// TIA Portal project "Assembler" (V17)

(* hardware
DEVICE "S7-1500/ET200MP station_1"  S7-1500 station
   slot 0: "Rail_0"  Rack  6ES7 590-1***0-0AA0
   slot 1: "PLC_1"  CPU 1511-1 PN  6ES7 511-1AK02-0AB0  V2.9
      slot 3: "CPU display_1"  6ES7591-1AA00-0AA0
      slot 32768: "PROFINET interface_1"  X1
         slot 32769: "Port_1"  X1 P1
         slot 32770: "Port_2"  X1 P2
      slot 34817: "Virtual CP interface port_1"  Virtual CP interface port  Virtual CP interface port
   slot 2: "DI 32x24VDC BA_1"  DI 32x24VDC BA  6ES7 521-1BL10-0AA0  V1.1
   slot 3: "DQ 32x24VDC/0.5A BA_1"  DQ 32x24VDC/0.5A BA  6ES7 522-1BL10-0AA0  V1.1
   slot 4: "AI 8xU/I/R/RTD BA_1"  AI 8xU/I/R/RTD BA  6ES7 531-7QF00-0AB0  V1.0
   slot 5: "AQ 8xU/I HS_1"  AQ 8xU/I HS  6ES7 532-5HF00-0AB0  V2.1
DEVICE "HMI_1"  KTP700 Basic PN
   slot 0: "HMI_1"  KTP700 Basic PN  6AV2 123-2GB03-0AX0  17.0.0.0
   slot 1: "HMI_RT_1"  KTP700 Basic PN  6AV2 123-2GB03-0AX0  17.0.0.0
   slot 5: "HMI_1.IE_CP_1"  PROFINET Interface  17.0.0.0
      slot 1: "PROFINET Interface_1"  PROFINET Interface
         slot 1: "Port_1"  Port
*)

// ===== PLC "PLC_1"  CPU 1511-1 PN =====

VAR_GLOBAL   // PLC tag table "Flanker"
   "Flank1" AT %M0.0 : Bool;
   "Flank2" AT %M0.1 : Bool;
   "Flank3" AT %M0.2 : Bool;
   "Flank4" AT %M0.3 : Bool;
   "Flank5" AT %M0.4 : Bool;
   "Flank6" AT %M0.5 : Bool;
   "Flank7" AT %M0.6 : Bool;
   "Flank8" AT %M0.7 : Bool;
   "Flank9" AT %M1.0 : Bool;
   "Flank10" AT %M1.1 : Bool;
END_VAR

VAR_GLOBAL   // PLC tag table "IO"
   "Lid at place" AT %I0.3 : Bool;
   "Lid clamped" AT %I0.4 : Bool;
   "Pos. at limit (lids)" AT %I0.5 : Bool;
   "Base at place" AT %I0.6 : Bool;
   "Base clamped" AT %I0.7 : Bool;
   "Pos. at limit (bases)" AT %I1.0 : Bool;
   "Part leaving scale" AT %I2.5 : Bool;
   "Start" AT %I1.2 : Bool;
   "Reset" AT %I1.3 : Bool;
   "Stop" AT %I1.4 : Bool;
   "Emergency stop" AT %I1.5 : Bool;
   "Manual" AT %I1.6 : Bool;
   "Auto" AT %I1.7 : Bool;
   "FACTORY I/O (Running)" AT %I2.0 : Bool;
   "Two-Axis Pick & Place 1 (Rotating)" AT %I2.1 : Bool;
   "Two-Axis Pick & Place 1 (Item Detected)" AT %I2.2 : Bool;
   "Two-Axis Pick & Place 1 (Gripper Rotating)" AT %I2.3 : Bool;
   "Part at scale" AT %I2.4 : Bool;
   "Bases emitter" AT %Q0.1 : Bool;
   "Lids emitter" AT %Q0.2 : Bool;
   "Lids conveyor" AT %Q0.3 : Bool;
   "Clamp lid" AT %Q0.4 : Bool;
   "Pos. raise (lids)" AT %Q0.5 : Bool;
   "Bases conveyor" AT %Q0.6 : Bool;
   "Clamp base" AT %Q0.7 : Bool;
   "Pos. raise (bases)" AT %Q1.0 : Bool;
   "Start light" AT %Q1.1 : Bool;
   "Reset light" AT %Q1.2 : Bool;
   "Stop light" AT %Q1.3 : Bool;
   "Remover 1" AT %Q1.4 : Bool;
   "Remover 2" AT %Q1.5 : Bool;
   "Conveyor Scale 0 (+)" AT %Q1.6 : Bool;
   "Conveyor Scale 0 (-)" AT %Q1.7 : Bool;
   "Two-Axis Pick & Place 1 (Grab)" AT %Q2.0 : Bool;
   "Two-Axis Pick & Place 1 Rotate CW" AT %Q2.1 : Bool;
   "Two-Axis Pick & Place 1 Gripper CW" AT %Q2.2 : Bool;
   "Two-Axis Pick & Place 1 Rotate CCW" AT %Q2.3 : Bool;
   "Two-Axis Pick & Place 1 Gripper CCW" AT %Q2.4 : Bool;
   "Conveyor Scale 0 Weight (V)" AT %IW30 : Int;
   "Two-Axis Pick & Place 1 X Position (V)" AT %IW32 : Int;
   "Two-Axis Pick & Place 1 Z Position (V)" AT %IW34 : Int;
   "Vision Sensor 0" AT %IW36 : Int;
   "Vision Sensor 1" AT %IW38 : Int;
   "Total Counter" AT %QW30 : Int;
   "Two-Axis Pick & Place 1 X Set Point (V)" AT %QW32 : Int;
   "Two-Axis Pick & Place 1 Z Set Point (V)" AT %QW34 : Int;
   "Weight" AT %QW36 : Int;
   "GB&GL" AT %QW38 : Int;
   "BB&BL" AT %QW40 : Int;
   "GB&BL" AT %QW42 : Int;
   "BB&GL" AT %QW44 : Int;
   "Part leaving" AT %I1.1 : Bool;
END_VAR

DATA_BLOCK "Skallering"   // DB1
{ S7_Optimized_Access := 'TRUE' }
VERSION : 0.1
   VAR
      IN : Struct
         "X är" : Struct
            "Norm min" : Int;
            "Norm max" : Int := 27648;
            "Norm value" : Real;
            "Scale min" : Real;
            "Scale max" : Real := 1.125;
            "X ärvärde" : Real;
         END_STRUCT;
         "Z är" : Struct
            "Norm min" : Int;
            "Norm max" : Int := 27648;
            "Norm value" : Real;
            "Scale min" : Real;
            "Scale max" : Real := 0.625;
            "Z ärvärde" : Real;
         END_STRUCT;
         "V är" : Struct
            "Norm min" : Int;
            "Norm max" : Int := 27648;
            "Norm value" : Real;
            "Scale min" : Int;
            "Scale max" : Int := 20;
            "V ärvärde" : Int;
         END_STRUCT;
      END_STRUCT;
      UT : Struct
         "X bör" : Struct
            "Norm min" : Real;
            "Norm max" : Real := 1.125;
            "Norm value" : Real;
            "Scale min" : Int;
            "Scale max" : Int := 27648;
            "X börvärde" : Real;
         END_STRUCT;
         "Z bör" : Struct
            "Norm min" : Real;
            "Norm max" : Real := 0.625;
            "Norm value" : Real;
            "Scale min" : Int;
            "Scale max" : Int := 27648;
            "Z börvärde" : Real;
         END_STRUCT;
      END_STRUCT;
   END_VAR
BEGIN
END_DATA_BLOCK

DATA_BLOCK "Hmi_Data"   // DB2
{ S7_Optimized_Access := 'TRUE' }
VERSION : 0.1
   VAR
      Start : Bool;
      Stop : Bool;
      Reset : Bool;
      Sekvensord : Int;
      "Reset Sekvens" : Int;
      Beställning : Int;
      "Antal Producedrade" : Int;
      Order : Bool;
   END_VAR
BEGIN
END_DATA_BLOCK

DATA_BLOCK "ManualData"   // DB12
{ S7_Optimized_Access := 'TRUE' }
VERSION : 0.1
   VAR
      Manual10 : Struct
         R : Bool;
         S : Bool;
         "R light" : Bool;
         "S light" : Bool;
      END_STRUCT;
      Manual11 : Struct
         R : Bool;
         S : Bool;
         "R light" : Bool;
         "S light" : Bool;
      END_STRUCT;
      Manual12 : Struct
         R : Bool;
         S : Bool;
         "R light" : Bool;
         "S light" : Bool;
      END_STRUCT;
      Manual13 : Struct
         R : Bool;
         S : Bool;
         "R light" : Bool;
         "S light" : Bool;
      END_STRUCT;
      Manual14 : Struct
         R : Bool;
         S : Bool;
         "R light" : Bool;
         "S light" : Bool;
      END_STRUCT;
      Manual15 : Struct
         R : Bool;
         S : Bool;
         "R light" : Bool;
         "S light" : Bool;
      END_STRUCT;
      Manual16 : Struct
         R : Bool;
         S : Bool;
         "R light" : Bool;
         "S light" : Bool;
      END_STRUCT;
      Manual17 : Struct
         R : Bool;
         S : Bool;
         "R light" : Bool;
         "S light" : Bool;
      END_STRUCT;
      Manual18 : Struct
         R : Bool;
         S : Bool;
         "R light" : Bool;
         "S light" : Bool;
      END_STRUCT;
      Manual19 : Struct
         R : Bool;
         S : Bool;
         "R light" : Bool;
         "S light" : Bool;
      END_STRUCT;
      ManualRobot : Struct
         "X+" : Bool;
         "X-" : Bool;
         "Z+" : Bool;
         "Z-" : Bool;
      END_STRUCT;
      "Hämta Z" : Real;
      "Ovan Hämta Z" : Real;
      "Ovan Lämna X" : Real;
      "Lämna X" : Real;
      "Spela in Hämta" : Bool;
      "Spela in Ovan Hämta" : Bool;
      "Spela in Ovan Lämna" : Bool;
      "Spela in Lämna" : Bool;
   END_VAR
BEGIN
END_DATA_BLOCK

// folder: System blocks/Program resources

DATA_BLOCK "IEC_Timer_0_DB"   // DB3
{ S7_Optimized_Access := 'TRUE' }
AUTHOR : Simatic
FAMILY : IEC
NAME : IEC_TMR
VERSION : 1.0
// stored: InstanceOfName IEC_TIMER
"IEC_TIMER"
BEGIN
END_DATA_BLOCK

DATA_BLOCK "IEC_Timer_0_DB_2"   // DB4
{ S7_Optimized_Access := 'TRUE' }
AUTHOR : Simatic
FAMILY : IEC
NAME : IEC_TMR
VERSION : 1.0
// stored: InstanceOfName IEC_TIMER
"IEC_TIMER"
BEGIN
END_DATA_BLOCK

DATA_BLOCK "IEC_Timer_0_DB_3"   // DB5
{ S7_Optimized_Access := 'TRUE' }
AUTHOR : Simatic
FAMILY : IEC
NAME : IEC_TMR
VERSION : 1.0
// stored: InstanceOfName IEC_TIMER
"IEC_TIMER"
BEGIN
END_DATA_BLOCK

DATA_BLOCK "IEC_Timer_0_DB_1"   // DB6
{ S7_Optimized_Access := 'TRUE' }
AUTHOR : Simatic
FAMILY : IEC
NAME : IEC_TMR
VERSION : 1.0
// stored: InstanceOfName IEC_TIMER
"IEC_TIMER"
BEGIN
END_DATA_BLOCK

DATA_BLOCK "IEC_Timer_0_DB_4"   // DB7
{ S7_Optimized_Access := 'TRUE' }
AUTHOR : Simatic
FAMILY : IEC
NAME : IEC_TMR
VERSION : 1.0
// stored: InstanceOfName IEC_TIMER
"IEC_TIMER"
BEGIN
END_DATA_BLOCK

DATA_BLOCK "IEC_Timer_0_DB_5"   // DB9
{ S7_Optimized_Access := 'TRUE' }
AUTHOR : Simatic
FAMILY : IEC
NAME : IEC_TMR
VERSION : 1.0
// stored: InstanceOfName IEC_TIMER
"IEC_TIMER"
BEGIN
END_DATA_BLOCK

DATA_BLOCK "IEC_Timer_0_DB_6"   // DB11
{ S7_Optimized_Access := 'TRUE' }
AUTHOR : Simatic
FAMILY : IEC
NAME : IEC_TMR
VERSION : 1.0
// stored: InstanceOfName IEC_TIMER
"IEC_TIMER"
BEGIN
END_DATA_BLOCK

// folder: (top level)

FUNCTION "Hmi" : Void   // FC1, LAD
{ S7_Optimized_Access := 'TRUE' }
VERSION : 0.1
   VAR_TEMP   // added for the SCL form of the ladder/FBD networks
      _w1 : Bool;
   END_VAR
BEGIN

REGION Network 1: Start
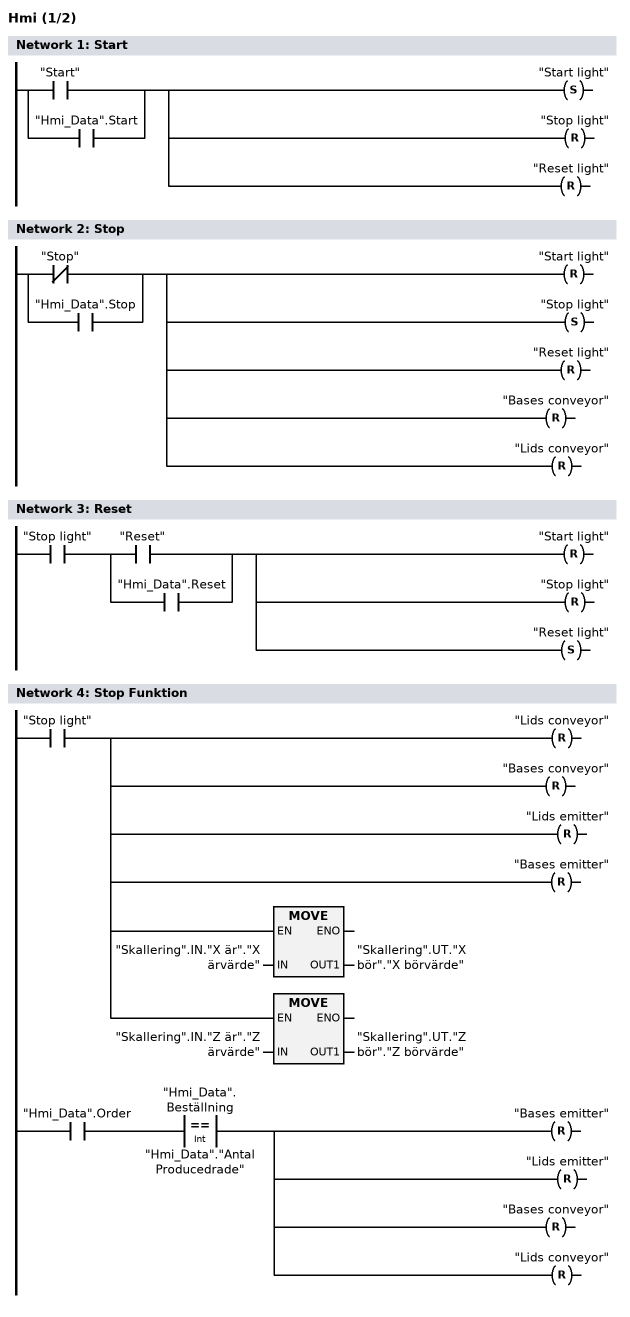
   RUNG wire#powerrail
      Contact( "Start" )
      wire#w1
      S_Coil( "Start light" )
   END_RUNG
   RUNG wire#powerrail
      Contact( "Hmi_Data".Start )
   END_RUNG wire#w1
   RUNG wire#w1
      R_Coil( "Stop light" )
   END_RUNG
   RUNG wire#w1
      R_Coil( "Reset light" )
   END_RUNG
   // the same network as SCL:
   IF "Start" OR "Hmi_Data".Start THEN
       "Start light" := TRUE;
       "Stop light" := FALSE;
       "Reset light" := FALSE;
   END_IF;
END_REGION

REGION Network 2: Stop
   RUNG wire#powerrail
      I_Contact( "Stop" )
      wire#w1
      R_Coil( "Start light" )
   END_RUNG
   RUNG wire#powerrail
      Contact( "Hmi_Data".Stop )
   END_RUNG wire#w1
   RUNG wire#w1
      S_Coil( "Stop light" )
   END_RUNG
   RUNG wire#w1
      R_Coil( "Reset light" )
   END_RUNG
   RUNG wire#w1
      R_Coil( "Bases conveyor" )
   END_RUNG
   RUNG wire#w1
      R_Coil( "Lids conveyor" )
   END_RUNG
   // the same network as SCL:
   IF NOT "Stop" OR "Hmi_Data".Stop THEN
       "Start light" := FALSE;
       "Stop light" := TRUE;
       "Reset light" := FALSE;
       "Bases conveyor" := FALSE;
       "Lids conveyor" := FALSE;
   END_IF;
END_REGION

REGION Network 3: Reset
   RUNG wire#powerrail
      Contact( "Stop light" )
      wire#w1
      Contact( "Reset" )
      wire#w2
      R_Coil( "Start light" )
   END_RUNG
   RUNG wire#w1
      Contact( "Hmi_Data".Reset )
   END_RUNG wire#w2
   RUNG wire#w2
      R_Coil( "Stop light" )
   END_RUNG
   RUNG wire#w2
      S_Coil( "Reset light" )
   END_RUNG
   // the same network as SCL:
   IF "Stop light" AND ("Reset" OR "Hmi_Data".Reset) THEN "Start light" := FALSE; END_IF;
   #_w1 := "Stop light" AND ("Reset" OR "Hmi_Data".Reset);
   IF #_w1 THEN
       "Stop light" := FALSE;
       "Reset light" := TRUE;
   END_IF;
END_REGION

REGION Network 4: Stop Funktion
   RUNG wire#powerrail
      Contact( "Stop light" )
      wire#w1
      R_Coil( "Lids conveyor" )
   END_RUNG
   RUNG wire#w1
      R_Coil( "Bases conveyor" )
   END_RUNG
   RUNG wire#w1
      R_Coil( "Lids emitter" )
   END_RUNG
   RUNG wire#w1
      R_Coil( "Bases emitter" )
   END_RUNG
   RUNG wire#w1
      Move(in := "Skallering".IN."X är"."X ärvärde", out1 => "Skallering".UT."X bör"."X börvärde")
   END_RUNG
   RUNG wire#w1
      Move(in := "Skallering".IN."Z är"."Z ärvärde", out1 => "Skallering".UT."Z bör"."Z börvärde")
   END_RUNG
   RUNG wire#powerrail
      Contact( "Hmi_Data".Order )
      { S7_Templates := "SrcType := Int" } EQ_Contact(in1 := "Hmi_Data".Beställning, in2 := "Hmi_Data"."Antal Producedrade")
      wire#w2
      R_Coil( "Bases emitter" )
   END_RUNG
   RUNG wire#w2
      R_Coil( "Lids emitter" )
   END_RUNG
   RUNG wire#w2
      R_Coil( "Bases conveyor" )
   END_RUNG
   RUNG wire#w2
      R_Coil( "Lids conveyor" )
   END_RUNG
   // the same network as SCL:
   IF "Stop light" THEN
       "Lids conveyor" := FALSE;
       "Bases conveyor" := FALSE;
       "Lids emitter" := FALSE;
       "Bases emitter" := FALSE;
       "Skallering".UT."X bör"."X börvärde" := "Skallering".IN."X är"."X ärvärde";
       "Skallering".UT."Z bör"."Z börvärde" := "Skallering".IN."Z är"."Z ärvärde";
   END_IF;
   IF "Hmi_Data".Order AND ("Hmi_Data".Beställning = "Hmi_Data"."Antal Producedrade") THEN
       "Bases emitter" := FALSE;
       "Lids emitter" := FALSE;
       "Bases conveyor" := FALSE;
       "Lids conveyor" := FALSE;
   END_IF;
END_REGION

REGION Network 5: Start Funktion
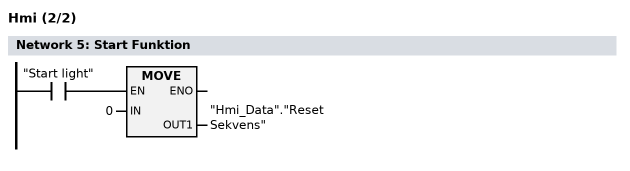
   RUNG wire#powerrail
      Contact( "Start light" )
      Move(in := 0, out1 => "Hmi_Data"."Reset Sekvens")
   END_RUNG
   // the same network as SCL:
   IF "Start light" THEN "Hmi_Data"."Reset Sekvens" := 0; END_IF;
END_REGION
END_FUNCTION

FUNCTION "IN Skallering" : Void   // FC2, LAD
{ S7_Optimized_Access := 'TRUE' }
VERSION : 0.1
BEGIN

REGION Network 1: Kontroll for X och Z ärvärde
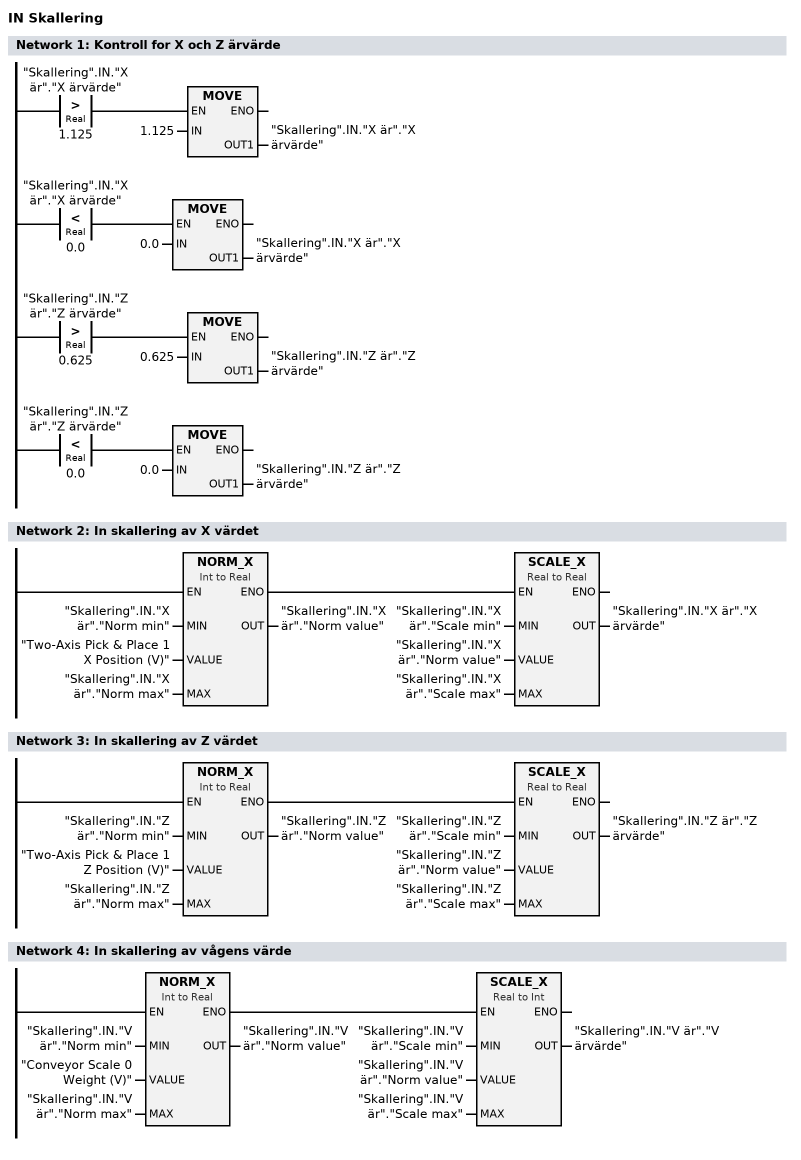
   RUNG wire#powerrail
      { S7_Templates := "SrcType := Real" } GT_Contact(in1 := "Skallering".IN."X är"."X ärvärde", in2 := 1.125)
      Move(in := 1.125, out1 => "Skallering".IN."X är"."X ärvärde")
   END_RUNG
   RUNG wire#powerrail
      { S7_Templates := "SrcType := Real" } LT_Contact(in1 := "Skallering".IN."X är"."X ärvärde", in2 := 0.0)
      Move(in := 0.0, out1 => "Skallering".IN."X är"."X ärvärde")
   END_RUNG
   RUNG wire#powerrail
      { S7_Templates := "SrcType := Real" } GT_Contact(in1 := "Skallering".IN."Z är"."Z ärvärde", in2 := 0.625)
      Move(in := 0.625, out1 => "Skallering".IN."Z är"."Z ärvärde")
   END_RUNG
   RUNG wire#powerrail
      { S7_Templates := "SrcType := Real" } LT_Contact(in1 := "Skallering".IN."Z är"."Z ärvärde", in2 := 0.0)
      Move(in := 0.0, out1 => "Skallering".IN."Z är"."Z ärvärde")
   END_RUNG
   // the same network as SCL:
   IF "Skallering".IN."X är"."X ärvärde" > 1.125 THEN "Skallering".IN."X är"."X ärvärde" := 1.125; END_IF;
   IF "Skallering".IN."X är"."X ärvärde" < 0.0 THEN "Skallering".IN."X är"."X ärvärde" := 0.0; END_IF;
   IF "Skallering".IN."Z är"."Z ärvärde" > 0.625 THEN "Skallering".IN."Z är"."Z ärvärde" := 0.625; END_IF;
   IF "Skallering".IN."Z är"."Z ärvärde" < 0.0 THEN "Skallering".IN."Z är"."Z ärvärde" := 0.0; END_IF;
END_REGION

REGION Network 2: In skallering av X värdet
   RUNG wire#powerrail
      { S7_Templates := "[SrcType := Int, DestType := Real]" } Normalize(min := "Skallering".IN."X är"."Norm min", value := "Two-Axis Pick & Place 1 X Position (V)", max := "Skallering".IN."X är"."Norm max", out => "Skallering".IN."X är"."Norm value")
      { S7_Templates := "[SrcType := Real, DestType := Real]" } Scale(min := "Skallering".IN."X är"."Scale min", value := "Skallering".IN."X är"."Norm value", max := "Skallering".IN."X är"."Scale max", out => "Skallering".IN."X är"."X ärvärde")
   END_RUNG
   // the same network as SCL:
   "Skallering".IN."X är"."Norm value" := NORM_X(MIN := "Skallering".IN."X är"."Norm min", VALUE := "Two-Axis Pick & Place 1 X Position (V)", MAX := "Skallering".IN."X är"."Norm max");
   "Skallering".IN."X är"."X ärvärde" := SCALE_X(MIN := "Skallering".IN."X är"."Scale min", VALUE := "Skallering".IN."X är"."Norm value", MAX := "Skallering".IN."X är"."Scale max");
END_REGION

REGION Network 3: In skallering av Z värdet
   RUNG wire#powerrail
      { S7_Templates := "[SrcType := Int, DestType := Real]" } Normalize(min := "Skallering".IN."Z är"."Norm min", value := "Two-Axis Pick & Place 1 Z Position (V)", max := "Skallering".IN."Z är"."Norm max", out => "Skallering".IN."Z är"."Norm value")
      { S7_Templates := "[SrcType := Real, DestType := Real]" } Scale(min := "Skallering".IN."Z är"."Scale min", value := "Skallering".IN."Z är"."Norm value", max := "Skallering".IN."Z är"."Scale max", out => "Skallering".IN."Z är"."Z ärvärde")
   END_RUNG
   // the same network as SCL:
   "Skallering".IN."Z är"."Norm value" := NORM_X(MIN := "Skallering".IN."Z är"."Norm min", VALUE := "Two-Axis Pick & Place 1 Z Position (V)", MAX := "Skallering".IN."Z är"."Norm max");
   "Skallering".IN."Z är"."Z ärvärde" := SCALE_X(MIN := "Skallering".IN."Z är"."Scale min", VALUE := "Skallering".IN."Z är"."Norm value", MAX := "Skallering".IN."Z är"."Scale max");
END_REGION

REGION Network 4: In skallering av vågens värde
   RUNG wire#powerrail
      { S7_Templates := "[SrcType := Int, DestType := Real]" } Normalize(min := "Skallering".IN."V är"."Norm min", value := "Conveyor Scale 0 Weight (V)", max := "Skallering".IN."V är"."Norm max", out => "Skallering".IN."V är"."Norm value")
      { S7_Templates := "[SrcType := Real, DestType := Int]" } Scale(min := "Skallering".IN."V är"."Scale min", value := "Skallering".IN."V är"."Norm value", max := "Skallering".IN."V är"."Scale max", out => "Skallering".IN."V är"."V ärvärde")
   END_RUNG
   // the same network as SCL:
   "Skallering".IN."V är"."Norm value" := NORM_X(MIN := "Skallering".IN."V är"."Norm min", VALUE := "Conveyor Scale 0 Weight (V)", MAX := "Skallering".IN."V är"."Norm max");
   "Skallering".IN."V är"."V ärvärde" := SCALE_X(MIN := "Skallering".IN."V är"."Scale min", VALUE := "Skallering".IN."V är"."Norm value", MAX := "Skallering".IN."V är"."Scale max");
END_REGION
END_FUNCTION

FUNCTION "UT Skallering" : Void   // FC3, LAD
{ S7_Optimized_Access := 'TRUE' }
VERSION : 0.1
BEGIN

REGION Network 1: Kontroll for X och Z börvärde
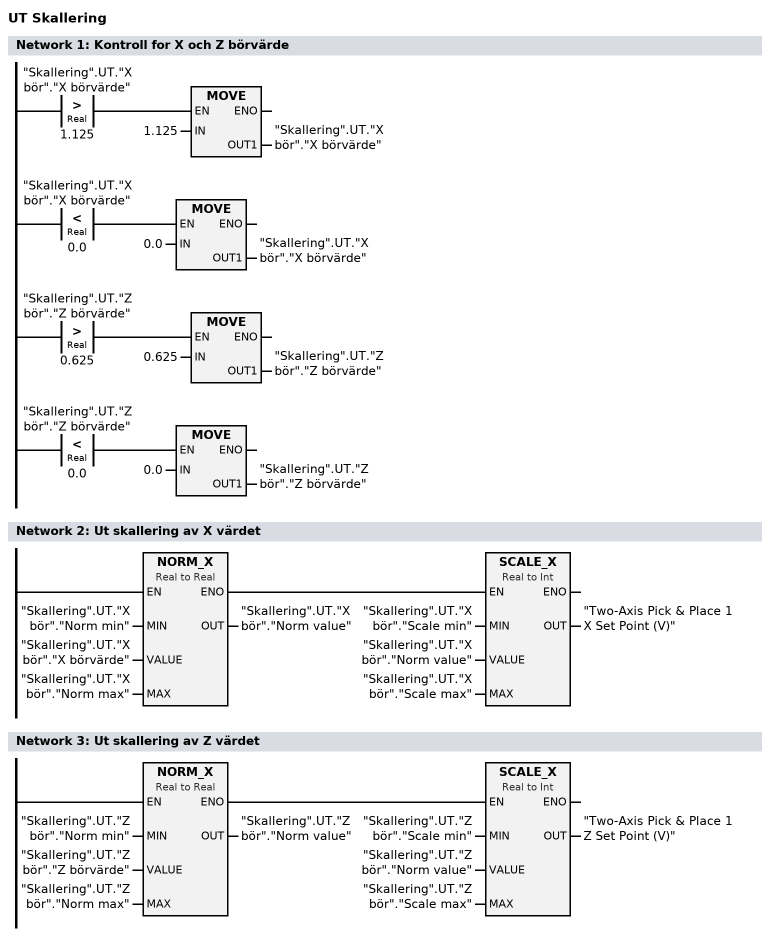
   RUNG wire#powerrail
      { S7_Templates := "SrcType := Real" } GT_Contact(in1 := "Skallering".UT."X bör"."X börvärde", in2 := 1.125)
      Move(in := 1.125, out1 => "Skallering".UT."X bör"."X börvärde")
   END_RUNG
   RUNG wire#powerrail
      { S7_Templates := "SrcType := Real" } LT_Contact(in1 := "Skallering".UT."X bör"."X börvärde", in2 := 0.0)
      Move(in := 0.0, out1 => "Skallering".UT."X bör"."X börvärde")
   END_RUNG
   RUNG wire#powerrail
      { S7_Templates := "SrcType := Real" } GT_Contact(in1 := "Skallering".UT."Z bör"."Z börvärde", in2 := 0.625)
      Move(in := 0.625, out1 => "Skallering".UT."Z bör"."Z börvärde")
   END_RUNG
   RUNG wire#powerrail
      { S7_Templates := "SrcType := Real" } LT_Contact(in1 := "Skallering".UT."Z bör"."Z börvärde", in2 := 0.0)
      Move(in := 0.0, out1 => "Skallering".UT."Z bör"."Z börvärde")
   END_RUNG
   // the same network as SCL:
   IF "Skallering".UT."X bör"."X börvärde" > 1.125 THEN
       "Skallering".UT."X bör"."X börvärde" := 1.125;
   END_IF;
   IF "Skallering".UT."X bör"."X börvärde" < 0.0 THEN "Skallering".UT."X bör"."X börvärde" := 0.0; END_IF;
   IF "Skallering".UT."Z bör"."Z börvärde" > 0.625 THEN
       "Skallering".UT."Z bör"."Z börvärde" := 0.625;
   END_IF;
   IF "Skallering".UT."Z bör"."Z börvärde" < 0.0 THEN "Skallering".UT."Z bör"."Z börvärde" := 0.0; END_IF;
END_REGION

REGION Network 2: Ut skallering av X värdet
   "Skallering".UT."X bör"."Norm value" := NORM_X(MIN := "Skallering".UT."X bör"."Norm min", VALUE := "Skallering".UT."X bör"."X börvärde", MAX := "Skallering".UT."X bör"."Norm max");
   "Two-Axis Pick & Place 1 X Set Point (V)" := SCALE_X(MIN := "Skallering".UT."X bör"."Scale min", VALUE := "Skallering".UT."X bör"."Norm value", MAX := "Skallering".UT."X bör"."Scale max");
END_REGION

REGION Network 3: Ut skallering av Z värdet
   "Skallering".UT."Z bör"."Norm value" := NORM_X(MIN := "Skallering".UT."Z bör"."Norm min", VALUE := "Skallering".UT."Z bör"."Z börvärde", MAX := "Skallering".UT."Z bör"."Norm max");
   "Two-Axis Pick & Place 1 Z Set Point (V)" := SCALE_X(MIN := "Skallering".UT."Z bör"."Scale min", VALUE := "Skallering".UT."Z bör"."Norm value", MAX := "Skallering".UT."Z bör"."Scale max");
END_REGION
END_FUNCTION

FUNCTION "Sekvens" : Void   // FC4, LAD
{ S7_Optimized_Access := 'TRUE' }
VERSION : 0.1
   VAR_TEMP   // added for the SCL form of the ladder/FBD networks
      _w1 : Bool;
      _w2 : Bool;
      _w3 : Bool;
      _w4 : Bool;
      _w5 : Bool;
   END_VAR
BEGIN

REGION Network 1: Sekvens 0: Sätta igång emitters och conveyors
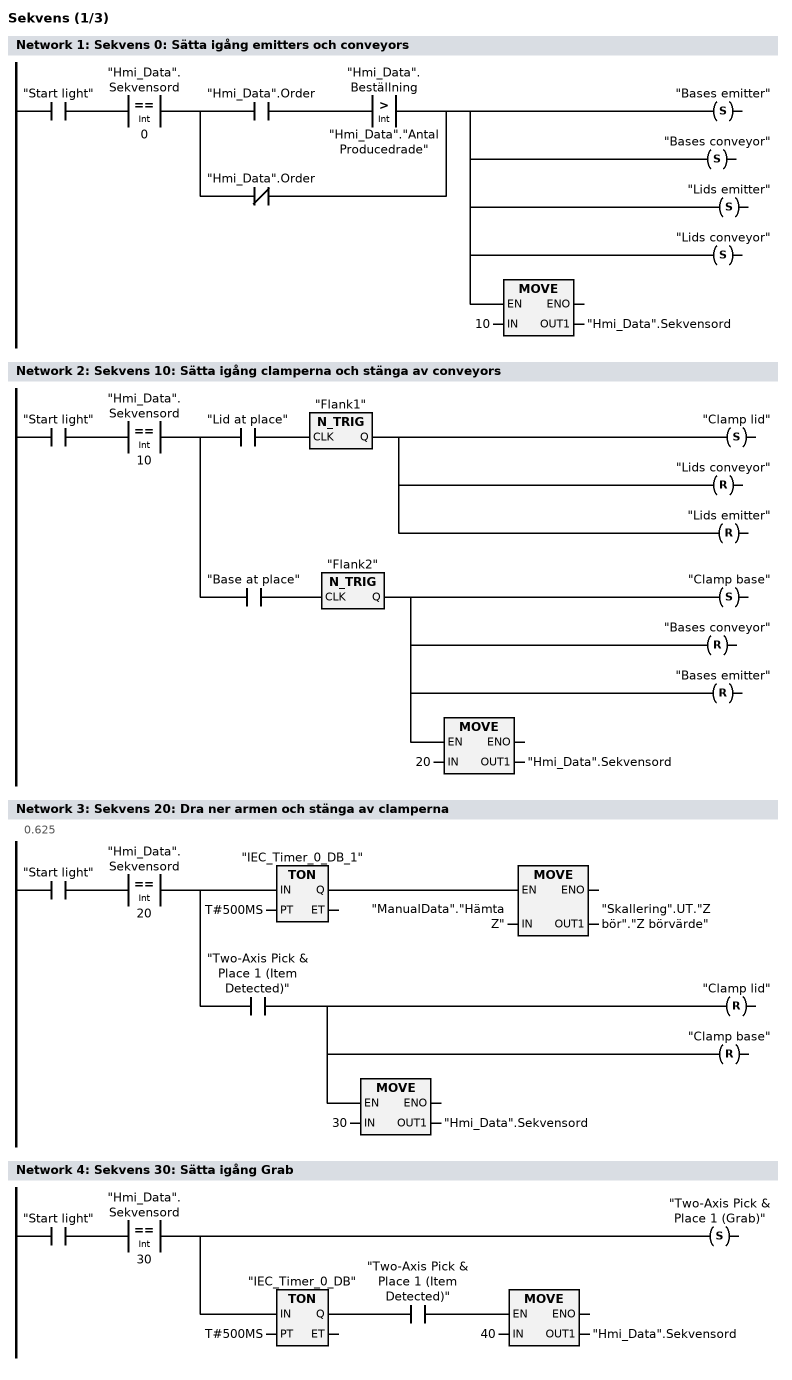
   RUNG wire#powerrail
      Contact( "Start light" )
      { S7_Templates := "SrcType := Int" } EQ_Contact(in1 := "Hmi_Data".Sekvensord, in2 := 0)
      wire#w1
      Contact( "Hmi_Data".Order )
      { S7_Templates := "SrcType := Int" } GT_Contact(in1 := "Hmi_Data".Beställning, in2 := "Hmi_Data"."Antal Producedrade")
      wire#w2
      S_Coil( "Bases emitter" )
   END_RUNG
   RUNG wire#w1
      I_Contact( "Hmi_Data".Order )
   END_RUNG wire#w2
   RUNG wire#w2
      S_Coil( "Bases conveyor" )
   END_RUNG
   RUNG wire#w2
      S_Coil( "Lids emitter" )
   END_RUNG
   RUNG wire#w2
      S_Coil( "Lids conveyor" )
   END_RUNG
   RUNG wire#w2
      Move(in := 10, out1 => "Hmi_Data".Sekvensord)
   END_RUNG
   // the same network as SCL:
   IF "Start light" AND ("Hmi_Data".Sekvensord = 0) AND (("Hmi_Data".Order AND ("Hmi_Data".Beställning > "Hmi_Data"."Antal Producedrade")) OR NOT "Hmi_Data".Order) THEN
       "Bases emitter" := TRUE;
       "Bases conveyor" := TRUE;
       "Lids emitter" := TRUE;
       "Lids conveyor" := TRUE;
       "Hmi_Data".Sekvensord := 10;
   END_IF;
END_REGION

REGION Network 2: Sekvens 10: Sätta igång clamperna och stänga av conveyors
   RUNG wire#powerrail
      Contact( "Start light" )
      { S7_Templates := "SrcType := Int" } EQ_Contact(in1 := "Hmi_Data".Sekvensord, in2 := 10)
      wire#w1
      Contact( "Lid at place" )
      N_Trig( "Flank1" )
      wire#w2
      S_Coil( "Clamp lid" )
   END_RUNG
   RUNG wire#w2
      R_Coil( "Lids conveyor" )
   END_RUNG
   RUNG wire#w2
      R_Coil( "Lids emitter" )
   END_RUNG
   RUNG wire#w1
      Contact( "Base at place" )
      N_Trig( "Flank2" )
      wire#w3
      S_Coil( "Clamp base" )
   END_RUNG
   RUNG wire#w3
      R_Coil( "Bases conveyor" )
   END_RUNG
   RUNG wire#w3
      R_Coil( "Bases emitter" )
   END_RUNG
   RUNG wire#w3
      Move(in := 20, out1 => "Hmi_Data".Sekvensord)
   END_RUNG
   // the same network as SCL:
   #_w1 := "Start light" AND ("Hmi_Data".Sekvensord = 10);
   #_w2 := #_w1 AND "Lid at place";
   #_w3 := NOT #_w2 AND "Flank1";   // falling edge
   "Flank1" := #_w2;
   IF #_w3 THEN
       "Clamp lid" := TRUE;
       "Lids conveyor" := FALSE;
       "Lids emitter" := FALSE;
   END_IF;
   #_w4 := #_w1 AND "Base at place";
   #_w5 := NOT #_w4 AND "Flank2";   // falling edge
   "Flank2" := #_w4;
   IF #_w5 THEN
       "Clamp base" := TRUE;
       "Bases conveyor" := FALSE;
       "Bases emitter" := FALSE;
       "Hmi_Data".Sekvensord := 20;
   END_IF;
END_REGION

REGION Network 3: Sekvens 20: Dra ner armen och stänga av clamperna
   // 0.625
   #_w1 := "Start light" AND ("Hmi_Data".Sekvensord = 20);
   "IEC_Timer_0_DB_1".TON(IN := #_w1, PT := T#500MS);
   IF "IEC_Timer_0_DB_1".Q THEN "Skallering".UT."Z bör"."Z börvärde" := "ManualData"."Hämta Z"; END_IF;
   IF #_w1 AND "Two-Axis Pick & Place 1 (Item Detected)" THEN
       "Clamp lid" := FALSE;
       "Clamp base" := FALSE;
       "Hmi_Data".Sekvensord := 30;
   END_IF;
END_REGION

REGION Network 4: Sekvens 30: Sätta igång Grab
   #_w1 := "Start light" AND ("Hmi_Data".Sekvensord = 30);
   IF #_w1 THEN "Two-Axis Pick & Place 1 (Grab)" := TRUE; END_IF;
   "IEC_Timer_0_DB".TON(IN := #_w1, PT := T#500MS);
   IF "IEC_Timer_0_DB".Q AND "Two-Axis Pick & Place 1 (Item Detected)" THEN
       "Hmi_Data".Sekvensord := 40;
   END_IF;
END_REGION

REGION Network 5: Sekvens 40: Dra up armen
   // 0.0
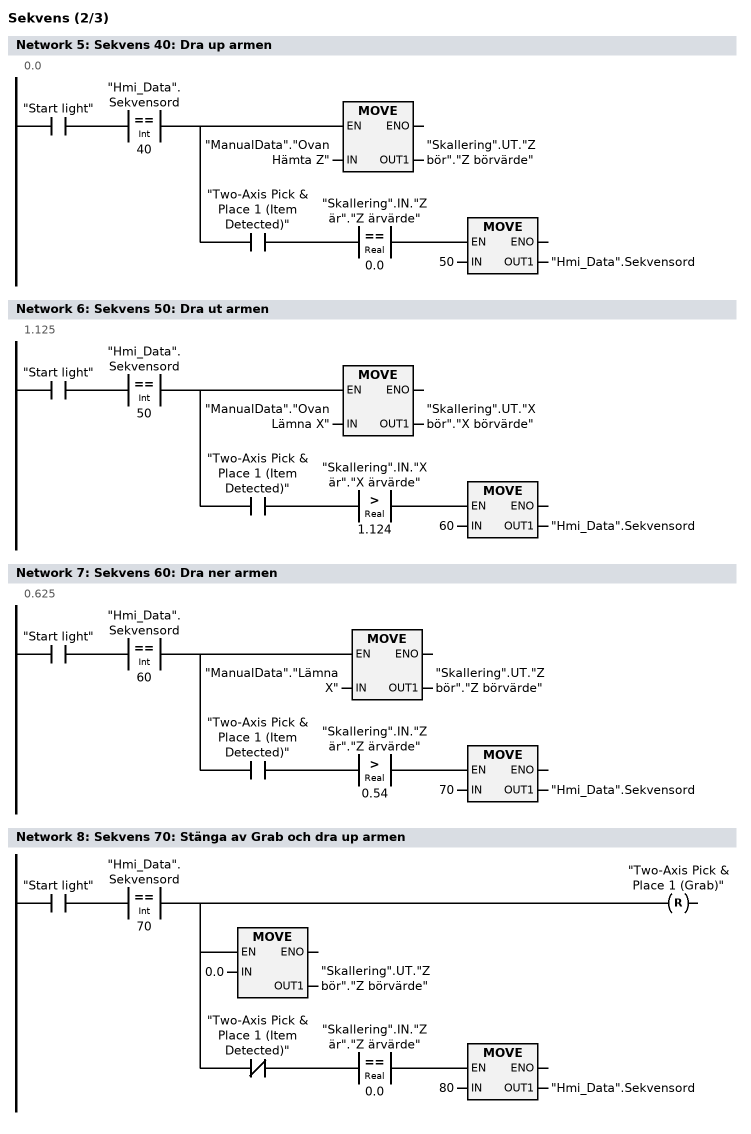
   RUNG wire#powerrail
      Contact( "Start light" )
      { S7_Templates := "SrcType := Int" } EQ_Contact(in1 := "Hmi_Data".Sekvensord, in2 := 40)
      wire#w1
      Move(in := "ManualData"."Ovan Hämta Z", out1 => "Skallering".UT."Z bör"."Z börvärde")
   END_RUNG
   RUNG wire#w1
      Contact( "Two-Axis Pick & Place 1 (Item Detected)" )
      { S7_Templates := "SrcType := Real" } EQ_Contact(in1 := "Skallering".IN."Z är"."Z ärvärde", in2 := 0.0)
      Move(in := 50, out1 => "Hmi_Data".Sekvensord)
   END_RUNG
   // the same network as SCL:
   #_w1 := "Start light" AND ("Hmi_Data".Sekvensord = 40);
   IF #_w1 THEN "Skallering".UT."Z bör"."Z börvärde" := "ManualData"."Ovan Hämta Z"; END_IF;
   IF #_w1 AND "Two-Axis Pick & Place 1 (Item Detected)" AND ("Skallering".IN."Z är"."Z ärvärde" = 0.0) THEN
       "Hmi_Data".Sekvensord := 50;
   END_IF;
END_REGION

REGION Network 6: Sekvens 50: Dra ut armen
   // 1.125
   RUNG wire#powerrail
      Contact( "Start light" )
      { S7_Templates := "SrcType := Int" } EQ_Contact(in1 := "Hmi_Data".Sekvensord, in2 := 50)
      wire#w1
      Move(in := "ManualData"."Ovan Lämna X", out1 => "Skallering".UT."X bör"."X börvärde")
   END_RUNG
   RUNG wire#w1
      Contact( "Two-Axis Pick & Place 1 (Item Detected)" )
      { S7_Templates := "SrcType := Real" } GT_Contact(in1 := "Skallering".IN."X är"."X ärvärde", in2 := 1.124)
      Move(in := 60, out1 => "Hmi_Data".Sekvensord)
   END_RUNG
   // the same network as SCL:
   #_w1 := "Start light" AND ("Hmi_Data".Sekvensord = 50);
   IF #_w1 THEN "Skallering".UT."X bör"."X börvärde" := "ManualData"."Ovan Lämna X"; END_IF;
   IF #_w1 AND "Two-Axis Pick & Place 1 (Item Detected)" AND ("Skallering".IN."X är"."X ärvärde" > 1.124) THEN
       "Hmi_Data".Sekvensord := 60;
   END_IF;
END_REGION

REGION Network 7: Sekvens 60: Dra ner armen
   // 0.625
   RUNG wire#powerrail
      Contact( "Start light" )
      { S7_Templates := "SrcType := Int" } EQ_Contact(in1 := "Hmi_Data".Sekvensord, in2 := 60)
      wire#w1
      Move(in := "ManualData"."Lämna X", out1 => "Skallering".UT."Z bör"."Z börvärde")
   END_RUNG
   RUNG wire#w1
      Contact( "Two-Axis Pick & Place 1 (Item Detected)" )
      { S7_Templates := "SrcType := Real" } GT_Contact(in1 := "Skallering".IN."Z är"."Z ärvärde", in2 := 0.54)
      Move(in := 70, out1 => "Hmi_Data".Sekvensord)
   END_RUNG
   // the same network as SCL:
   #_w1 := "Start light" AND ("Hmi_Data".Sekvensord = 60);
   IF #_w1 THEN "Skallering".UT."Z bör"."Z börvärde" := "ManualData"."Lämna X"; END_IF;
   IF #_w1 AND "Two-Axis Pick & Place 1 (Item Detected)" AND ("Skallering".IN."Z är"."Z ärvärde" > 0.54) THEN
       "Hmi_Data".Sekvensord := 70;
   END_IF;
END_REGION

REGION Network 8: Sekvens 70: Stänga av Grab och dra up armen
   RUNG wire#powerrail
      Contact( "Start light" )
      { S7_Templates := "SrcType := Int" } EQ_Contact(in1 := "Hmi_Data".Sekvensord, in2 := 70)
      wire#w1
      R_Coil( "Two-Axis Pick & Place 1 (Grab)" )
   END_RUNG
   RUNG wire#w1
      Move(in := 0.0, out1 => "Skallering".UT."Z bör"."Z börvärde")
   END_RUNG
   RUNG wire#w1
      I_Contact( "Two-Axis Pick & Place 1 (Item Detected)" )
      { S7_Templates := "SrcType := Real" } EQ_Contact(in1 := "Skallering".IN."Z är"."Z ärvärde", in2 := 0.0)
      Move(in := 80, out1 => "Hmi_Data".Sekvensord)
   END_RUNG
   // the same network as SCL:
   #_w1 := "Start light" AND ("Hmi_Data".Sekvensord = 70);
   IF #_w1 THEN
       "Two-Axis Pick & Place 1 (Grab)" := FALSE;
       "Skallering".UT."Z bör"."Z börvärde" := 0.0;
   END_IF;
   IF #_w1 AND NOT "Two-Axis Pick & Place 1 (Item Detected)" AND ("Skallering".IN."Z är"."Z ärvärde" = 0.0) THEN
       "Hmi_Data".Sekvensord := 80;
   END_IF;
END_REGION

REGION Network 9: Sekvens 80: Dra in armen och stätta igång Pos. raise, conveyors och stänga av emittrarna
   // 0.0
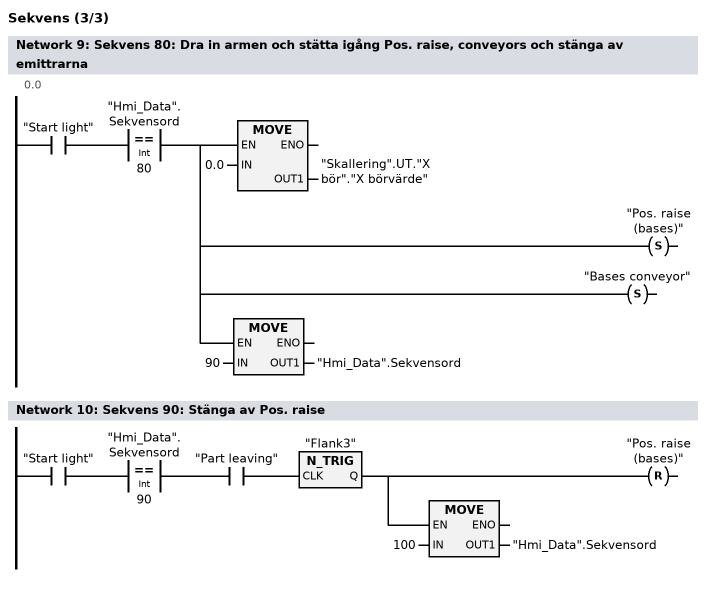
   RUNG wire#powerrail
      Contact( "Start light" )
      { S7_Templates := "SrcType := Int" } EQ_Contact(in1 := "Hmi_Data".Sekvensord, in2 := 80)
      wire#w1
      Move(in := 0.0, out1 => "Skallering".UT."X bör"."X börvärde")
   END_RUNG
   RUNG wire#w1
      S_Coil( "Pos. raise (bases)" )
   END_RUNG
   RUNG wire#w1
      S_Coil( "Bases conveyor" )
   END_RUNG
   RUNG wire#w1
      Move(in := 90, out1 => "Hmi_Data".Sekvensord)
   END_RUNG
   // the same network as SCL:
   IF "Start light" AND ("Hmi_Data".Sekvensord = 80) THEN
       "Skallering".UT."X bör"."X börvärde" := 0.0;
       "Pos. raise (bases)" := TRUE;
       "Bases conveyor" := TRUE;
       "Hmi_Data".Sekvensord := 90;
   END_IF;
END_REGION

REGION Network 10: Sekvens 90: Stänga av Pos. raise
   RUNG wire#powerrail
      Contact( "Start light" )
      { S7_Templates := "SrcType := Int" } EQ_Contact(in1 := "Hmi_Data".Sekvensord, in2 := 90)
      Contact( "Part leaving" )
      N_Trig( "Flank3" )
      wire#w1
      R_Coil( "Pos. raise (bases)" )
   END_RUNG
   RUNG wire#w1
      Move(in := 100, out1 => "Hmi_Data".Sekvensord)
   END_RUNG
   // the same network as SCL:
   #_w1 := "Start light" AND ("Hmi_Data".Sekvensord = 90) AND "Part leaving";
   #_w2 := NOT #_w1 AND "Flank3";   // falling edge
   "Flank3" := #_w1;
   IF #_w2 THEN
       "Pos. raise (bases)" := FALSE;
       "Hmi_Data".Sekvensord := 100;
   END_IF;
END_REGION
END_FUNCTION

FUNCTION "Raknare" : Void   // FC5, LAD
{ S7_Optimized_Access := 'TRUE' }
VERSION : 0.1
   VAR_TEMP   // added for the SCL form of the ladder/FBD networks
      _w1 : Bool;
      _w2 : Bool;
   END_VAR
BEGIN

REGION Network 1: Visa vågens värde
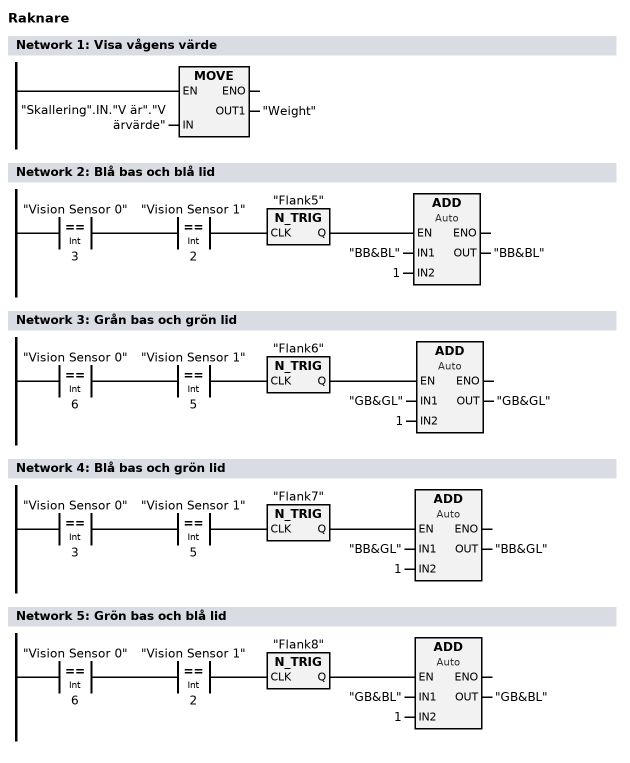
   RUNG wire#powerrail
      Move(in := "Skallering".IN."V är"."V ärvärde", out1 => "Weight")
   END_RUNG
   // the same network as SCL:
   "Weight" := "Skallering".IN."V är"."V ärvärde";
END_REGION

REGION Network 2: Blå bas och blå lid
   RUNG wire#powerrail
      { S7_Templates := "SrcType := Int" } EQ_Contact(in1 := "Vision Sensor 0", in2 := 3)
      { S7_Templates := "SrcType := Int" } EQ_Contact(in1 := "Vision Sensor 1", in2 := 2)
      N_Trig( "Flank5" )
      Add(in1 := "BB&BL", in2 := 1, out => "BB&BL")
   END_RUNG
   // the same network as SCL:
   #_w1 := ("Vision Sensor 0" = 3) AND ("Vision Sensor 1" = 2);
   #_w2 := NOT #_w1 AND "Flank5";   // falling edge
   "Flank5" := #_w1;
   IF #_w2 THEN "BB&BL" := "BB&BL" + 1; END_IF;
END_REGION

REGION Network 3: Grån bas och grön lid
   RUNG wire#powerrail
      { S7_Templates := "SrcType := Int" } EQ_Contact(in1 := "Vision Sensor 0", in2 := 6)
      { S7_Templates := "SrcType := Int" } EQ_Contact(in1 := "Vision Sensor 1", in2 := 5)
      N_Trig( "Flank6" )
      Add(in1 := "GB&GL", in2 := 1, out => "GB&GL")
   END_RUNG
   // the same network as SCL:
   #_w1 := ("Vision Sensor 0" = 6) AND ("Vision Sensor 1" = 5);
   #_w2 := NOT #_w1 AND "Flank6";   // falling edge
   "Flank6" := #_w1;
   IF #_w2 THEN "GB&GL" := "GB&GL" + 1; END_IF;
END_REGION

REGION Network 4: Blå bas och grön lid
   RUNG wire#powerrail
      { S7_Templates := "SrcType := Int" } EQ_Contact(in1 := "Vision Sensor 0", in2 := 3)
      { S7_Templates := "SrcType := Int" } EQ_Contact(in1 := "Vision Sensor 1", in2 := 5)
      N_Trig( "Flank7" )
      Add(in1 := "BB&GL", in2 := 1, out => "BB&GL")
   END_RUNG
   // the same network as SCL:
   #_w1 := ("Vision Sensor 0" = 3) AND ("Vision Sensor 1" = 5);
   #_w2 := NOT #_w1 AND "Flank7";   // falling edge
   "Flank7" := #_w1;
   IF #_w2 THEN "BB&GL" := "BB&GL" + 1; END_IF;
END_REGION

REGION Network 5: Grön bas och blå lid
   RUNG wire#powerrail
      { S7_Templates := "SrcType := Int" } EQ_Contact(in1 := "Vision Sensor 0", in2 := 6)
      { S7_Templates := "SrcType := Int" } EQ_Contact(in1 := "Vision Sensor 1", in2 := 2)
      N_Trig( "Flank8" )
      Add(in1 := "GB&BL", in2 := 1, out => "GB&BL")
   END_RUNG
   // the same network as SCL:
   #_w1 := ("Vision Sensor 0" = 6) AND ("Vision Sensor 1" = 2);
   #_w2 := NOT #_w1 AND "Flank8";   // falling edge
   "Flank8" := #_w1;
   IF #_w2 THEN "GB&BL" := "GB&BL" + 1; END_IF;
END_REGION
END_FUNCTION

FUNCTION "Reset Sekvens" : Void   // FC6, LAD
{ S7_Optimized_Access := 'TRUE' }
VERSION : 0.1
   VAR_TEMP   // added for the SCL form of the ladder/FBD networks
      _w1 : Bool;
   END_VAR
BEGIN

REGION Network 1: Sekvens 0: Skicka 10 till Reset Sekvensen om Grab är på annars skicka 100
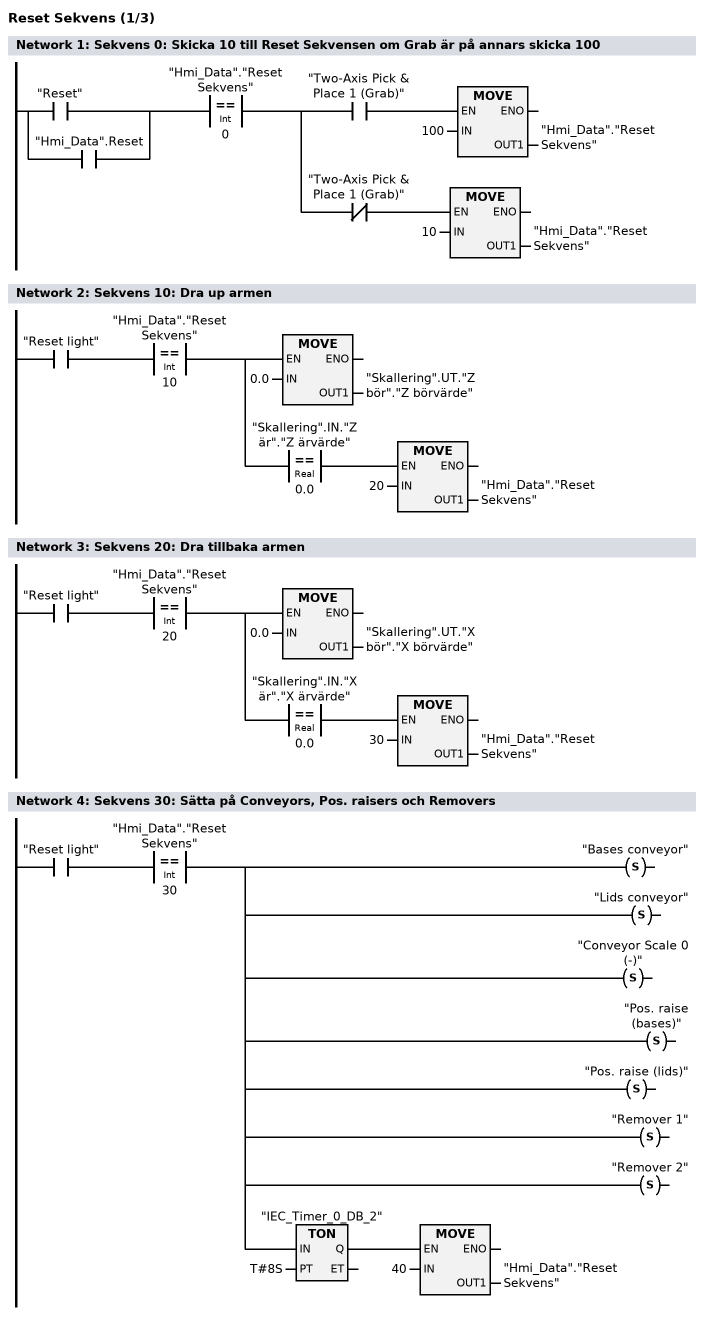
   RUNG wire#powerrail
      Contact( "Reset" )
      wire#w1
      { S7_Templates := "SrcType := Int" } EQ_Contact(in1 := "Hmi_Data"."Reset Sekvens", in2 := 0)
      wire#w2
      Contact( "Two-Axis Pick & Place 1 (Grab)" )
      Move(in := 100, out1 => "Hmi_Data"."Reset Sekvens")
   END_RUNG
   RUNG wire#powerrail
      Contact( "Hmi_Data".Reset )
   END_RUNG wire#w1
   RUNG wire#w2
      I_Contact( "Two-Axis Pick & Place 1 (Grab)" )
      Move(in := 10, out1 => "Hmi_Data"."Reset Sekvens")
   END_RUNG
   // the same network as SCL:
   #_w1 := ("Reset" OR "Hmi_Data".Reset) AND ("Hmi_Data"."Reset Sekvens" = 0);
   IF #_w1 AND "Two-Axis Pick & Place 1 (Grab)" THEN "Hmi_Data"."Reset Sekvens" := 100; END_IF;
   IF #_w1 AND NOT "Two-Axis Pick & Place 1 (Grab)" THEN "Hmi_Data"."Reset Sekvens" := 10; END_IF;
END_REGION

REGION Network 2: Sekvens 10: Dra up armen
   RUNG wire#powerrail
      Contact( "Reset light" )
      { S7_Templates := "SrcType := Int" } EQ_Contact(in1 := "Hmi_Data"."Reset Sekvens", in2 := 10)
      wire#w1
      Move(in := 0.0, out1 => "Skallering".UT."Z bör"."Z börvärde")
   END_RUNG
   RUNG wire#w1
      { S7_Templates := "SrcType := Real" } EQ_Contact(in1 := "Skallering".IN."Z är"."Z ärvärde", in2 := 0.0)
      Move(in := 20, out1 => "Hmi_Data"."Reset Sekvens")
   END_RUNG
   // the same network as SCL:
   #_w1 := "Reset light" AND ("Hmi_Data"."Reset Sekvens" = 10);
   IF #_w1 THEN "Skallering".UT."Z bör"."Z börvärde" := 0.0; END_IF;
   IF #_w1 AND ("Skallering".IN."Z är"."Z ärvärde" = 0.0) THEN "Hmi_Data"."Reset Sekvens" := 20; END_IF;
END_REGION

REGION Network 3: Sekvens 20: Dra tillbaka armen
   RUNG wire#powerrail
      Contact( "Reset light" )
      { S7_Templates := "SrcType := Int" } EQ_Contact(in1 := "Hmi_Data"."Reset Sekvens", in2 := 20)
      wire#w1
      Move(in := 0.0, out1 => "Skallering".UT."X bör"."X börvärde")
   END_RUNG
   RUNG wire#w1
      { S7_Templates := "SrcType := Real" } EQ_Contact(in1 := "Skallering".IN."X är"."X ärvärde", in2 := 0.0)
      Move(in := 30, out1 => "Hmi_Data"."Reset Sekvens")
   END_RUNG
   // the same network as SCL:
   #_w1 := "Reset light" AND ("Hmi_Data"."Reset Sekvens" = 20);
   IF #_w1 THEN "Skallering".UT."X bör"."X börvärde" := 0.0; END_IF;
   IF #_w1 AND ("Skallering".IN."X är"."X ärvärde" = 0.0) THEN "Hmi_Data"."Reset Sekvens" := 30; END_IF;
END_REGION

REGION Network 4: Sekvens 30: Sätta på Conveyors, Pos. raisers och Removers
   #_w1 := "Reset light" AND ("Hmi_Data"."Reset Sekvens" = 30);
   IF #_w1 THEN
       "Bases conveyor" := TRUE;
       "Lids conveyor" := TRUE;
       "Conveyor Scale 0 (-)" := TRUE;
       "Pos. raise (bases)" := TRUE;
       "Pos. raise (lids)" := TRUE;
       "Remover 1" := TRUE;
       "Remover 2" := TRUE;
   END_IF;
   "IEC_Timer_0_DB_2".TON(IN := #_w1, PT := T#8S);
   IF "IEC_Timer_0_DB_2".Q THEN "Hmi_Data"."Reset Sekvens" := 40; END_IF;
END_REGION

REGION Network 5: Sekvens 40: Stänga av Conveyors, Pos. raisers och Removers
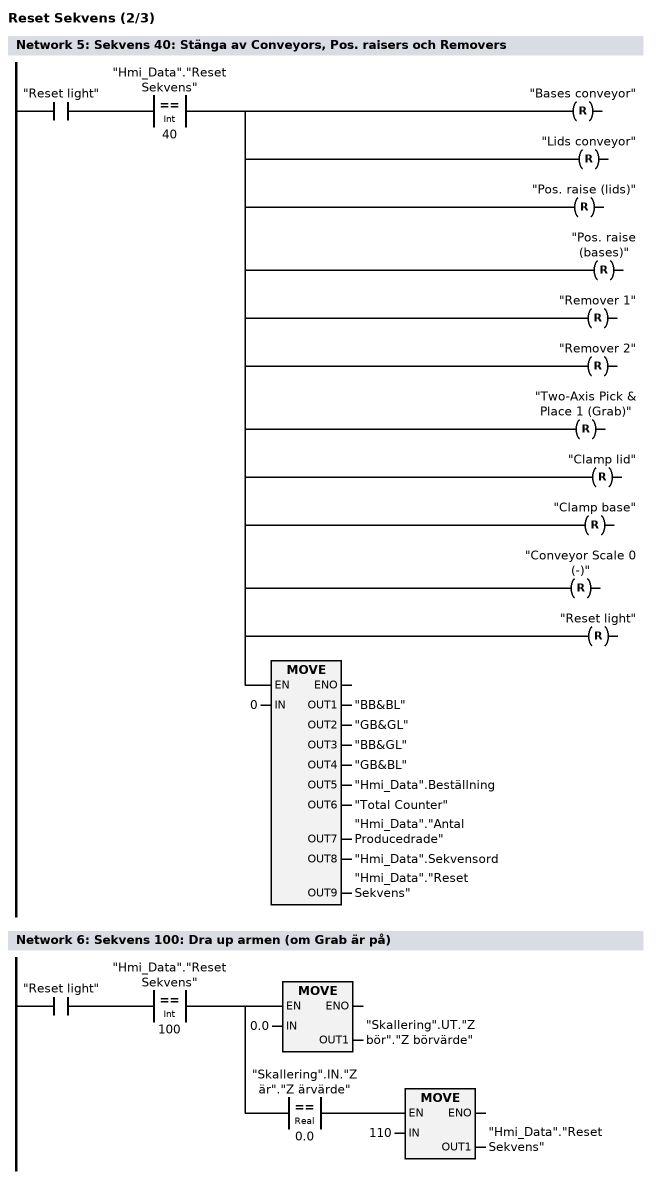
   RUNG wire#powerrail
      Contact( "Reset light" )
      { S7_Templates := "SrcType := Int" } EQ_Contact(in1 := "Hmi_Data"."Reset Sekvens", in2 := 40)
      wire#w1
      R_Coil( "Bases conveyor" )
   END_RUNG
   RUNG wire#w1
      R_Coil( "Lids conveyor" )
   END_RUNG
   RUNG wire#w1
      R_Coil( "Pos. raise (lids)" )
   END_RUNG
   RUNG wire#w1
      R_Coil( "Pos. raise (bases)" )
   END_RUNG
   RUNG wire#w1
      R_Coil( "Remover 1" )
   END_RUNG
   RUNG wire#w1
      R_Coil( "Remover 2" )
   END_RUNG
   RUNG wire#w1
      R_Coil( "Two-Axis Pick & Place 1 (Grab)" )
   END_RUNG
   RUNG wire#w1
      R_Coil( "Clamp lid" )
   END_RUNG
   RUNG wire#w1
      R_Coil( "Clamp base" )
   END_RUNG
   RUNG wire#w1
      R_Coil( "Conveyor Scale 0 (-)" )
   END_RUNG
   RUNG wire#w1
      R_Coil( "Reset light" )
   END_RUNG
   RUNG wire#w1
      Move(in := 0, out1 => "BB&BL", out2 => "GB&GL", out3 => "BB&GL", out4 => "GB&BL", out5 => "Hmi_Data".Beställning, out6 => "Total Counter", out7 => "Hmi_Data"."Antal Producedrade", out8 => "Hmi_Data".Sekvensord, out9 => "Hmi_Data"."Reset Sekvens")
   END_RUNG
   // the same network as SCL:
   IF "Reset light" AND ("Hmi_Data"."Reset Sekvens" = 40) THEN
       "Bases conveyor" := FALSE;
       "Lids conveyor" := FALSE;
       "Pos. raise (lids)" := FALSE;
       "Pos. raise (bases)" := FALSE;
       "Remover 1" := FALSE;
       "Remover 2" := FALSE;
       "Two-Axis Pick & Place 1 (Grab)" := FALSE;
       "Clamp lid" := FALSE;
       "Clamp base" := FALSE;
       "Conveyor Scale 0 (-)" := FALSE;
   END_IF;
   #_w1 := "Reset light" AND ("Hmi_Data"."Reset Sekvens" = 40);
   IF #_w1 THEN
       "Reset light" := FALSE;
       "BB&BL" := 0;
       "GB&GL" := 0;
       "BB&GL" := 0;
       "GB&BL" := 0;
       "Hmi_Data".Beställning := 0;
       "Total Counter" := 0;
       "Hmi_Data"."Antal Producedrade" := 0;
       "Hmi_Data".Sekvensord := 0;
       "Hmi_Data"."Reset Sekvens" := 0;
   END_IF;
END_REGION

REGION Network 6: Sekvens 100: Dra up armen (om Grab är på)
   RUNG wire#powerrail
      Contact( "Reset light" )
      { S7_Templates := "SrcType := Int" } EQ_Contact(in1 := "Hmi_Data"."Reset Sekvens", in2 := 100)
      wire#w1
      Move(in := 0.0, out1 => "Skallering".UT."Z bör"."Z börvärde")
   END_RUNG
   RUNG wire#w1
      { S7_Templates := "SrcType := Real" } EQ_Contact(in1 := "Skallering".IN."Z är"."Z ärvärde", in2 := 0.0)
      Move(in := 110, out1 => "Hmi_Data"."Reset Sekvens")
   END_RUNG
   // the same network as SCL:
   #_w1 := "Reset light" AND ("Hmi_Data"."Reset Sekvens" = 100);
   IF #_w1 THEN "Skallering".UT."Z bör"."Z börvärde" := 0.0; END_IF;
   IF #_w1 AND ("Skallering".IN."Z är"."Z ärvärde" = 0.0) THEN "Hmi_Data"."Reset Sekvens" := 110; END_IF;
END_REGION

REGION Network 7: Sekvens 110: Dra tillbaka armen (om Grab är på)
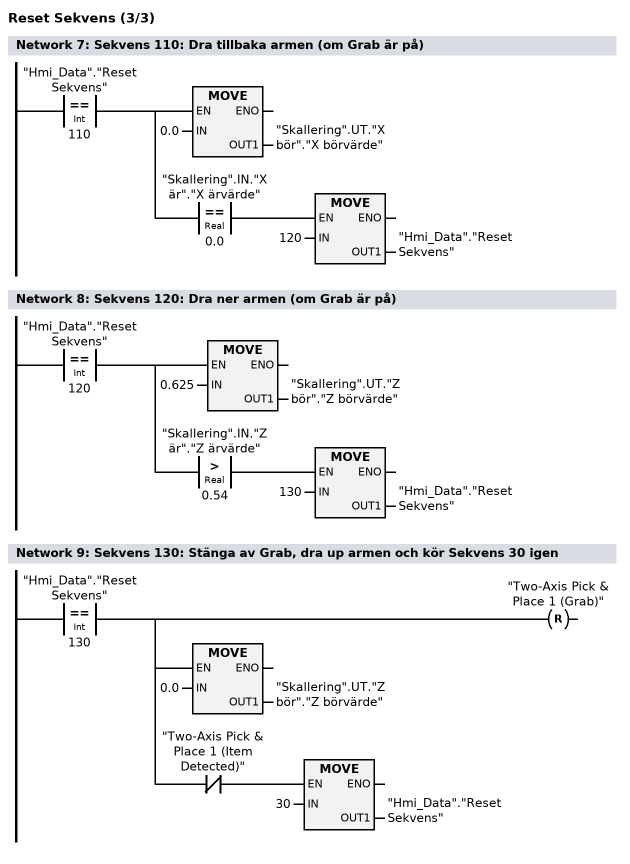
   RUNG wire#powerrail
      { S7_Templates := "SrcType := Int" } EQ_Contact(in1 := "Hmi_Data"."Reset Sekvens", in2 := 110)
      wire#w1
      Move(in := 0.0, out1 => "Skallering".UT."X bör"."X börvärde")
   END_RUNG
   RUNG wire#w1
      { S7_Templates := "SrcType := Real" } EQ_Contact(in1 := "Skallering".IN."X är"."X ärvärde", in2 := 0.0)
      Move(in := 120, out1 => "Hmi_Data"."Reset Sekvens")
   END_RUNG
   // the same network as SCL:
   #_w1 := "Hmi_Data"."Reset Sekvens" = 110;
   IF #_w1 THEN "Skallering".UT."X bör"."X börvärde" := 0.0; END_IF;
   IF #_w1 AND ("Skallering".IN."X är"."X ärvärde" = 0.0) THEN "Hmi_Data"."Reset Sekvens" := 120; END_IF;
END_REGION

REGION Network 8: Sekvens 120: Dra ner armen (om Grab är på)
   RUNG wire#powerrail
      { S7_Templates := "SrcType := Int" } EQ_Contact(in1 := "Hmi_Data"."Reset Sekvens", in2 := 120)
      wire#w1
      Move(in := 0.625, out1 => "Skallering".UT."Z bör"."Z börvärde")
   END_RUNG
   RUNG wire#w1
      { S7_Templates := "SrcType := Real" } GT_Contact(in1 := "Skallering".IN."Z är"."Z ärvärde", in2 := 0.54)
      Move(in := 130, out1 => "Hmi_Data"."Reset Sekvens")
   END_RUNG
   // the same network as SCL:
   #_w1 := "Hmi_Data"."Reset Sekvens" = 120;
   IF #_w1 THEN "Skallering".UT."Z bör"."Z börvärde" := 0.625; END_IF;
   IF #_w1 AND ("Skallering".IN."Z är"."Z ärvärde" > 0.54) THEN "Hmi_Data"."Reset Sekvens" := 130; END_IF;
END_REGION

REGION Network 9: Sekvens 130: Stänga av Grab, dra up armen och kör Sekvens 30 igen
   RUNG wire#powerrail
      { S7_Templates := "SrcType := Int" } EQ_Contact(in1 := "Hmi_Data"."Reset Sekvens", in2 := 130)
      wire#w1
      R_Coil( "Two-Axis Pick & Place 1 (Grab)" )
   END_RUNG
   RUNG wire#w1
      Move(in := 0.0, out1 => "Skallering".UT."Z bör"."Z börvärde")
   END_RUNG
   RUNG wire#w1
      I_Contact( "Two-Axis Pick & Place 1 (Item Detected)" )
      Move(in := 30, out1 => "Hmi_Data"."Reset Sekvens")
   END_RUNG
   // the same network as SCL:
   #_w1 := "Hmi_Data"."Reset Sekvens" = 130;
   IF #_w1 THEN
       "Two-Axis Pick & Place 1 (Grab)" := FALSE;
       "Skallering".UT."Z bör"."Z börvärde" := 0.0;
   END_IF;
   IF #_w1 AND NOT "Two-Axis Pick & Place 1 (Item Detected)" THEN "Hmi_Data"."Reset Sekvens" := 30; END_IF;
END_REGION
END_FUNCTION

FUNCTION "Vagen" : Void   // FC7, LAD
{ S7_Optimized_Access := 'TRUE' }
VERSION : 0.1
   VAR_TEMP   // added for the SCL form of the ladder/FBD networks
      _w1 : Bool;
   END_VAR
BEGIN

REGION Network 1: Sekvens 100: Stätta på scale conveyor och removern
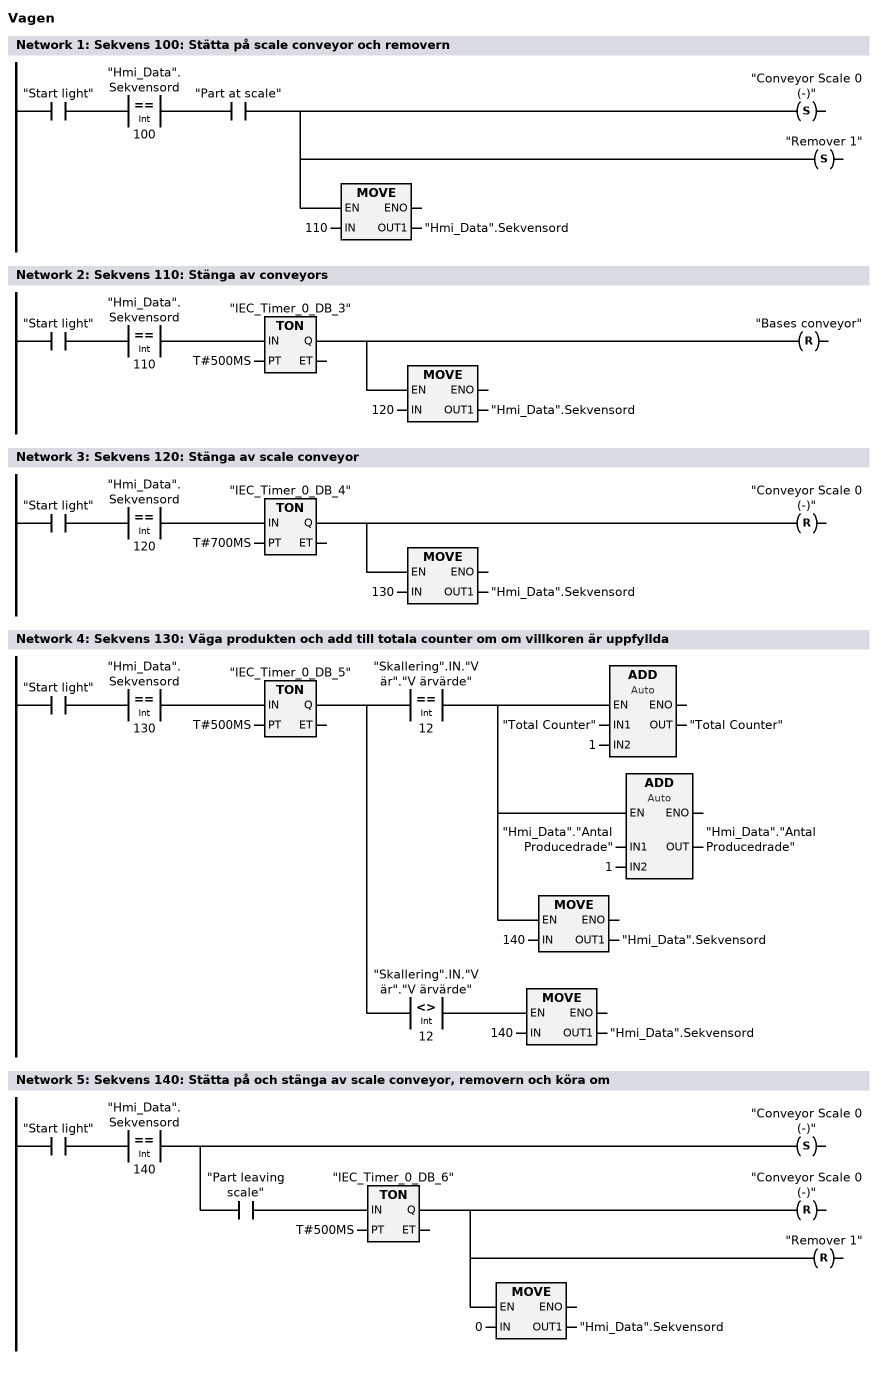
   RUNG wire#powerrail
      Contact( "Start light" )
      { S7_Templates := "SrcType := Int" } EQ_Contact(in1 := "Hmi_Data".Sekvensord, in2 := 100)
      Contact( "Part at scale" )
      wire#w1
      S_Coil( "Conveyor Scale 0 (-)" )
   END_RUNG
   RUNG wire#w1
      S_Coil( "Remover 1" )
   END_RUNG
   RUNG wire#w1
      Move(in := 110, out1 => "Hmi_Data".Sekvensord)
   END_RUNG
   // the same network as SCL:
   IF "Start light" AND ("Hmi_Data".Sekvensord = 100) AND "Part at scale" THEN
       "Conveyor Scale 0 (-)" := TRUE;
       "Remover 1" := TRUE;
       "Hmi_Data".Sekvensord := 110;
   END_IF;
END_REGION

REGION Network 2: Sekvens 110: Stänga av conveyors
   "IEC_Timer_0_DB_3".TON(IN := "Start light" AND ("Hmi_Data".Sekvensord = 110), PT := T#500MS);
   IF "IEC_Timer_0_DB_3".Q THEN
       "Bases conveyor" := FALSE;
       "Hmi_Data".Sekvensord := 120;
   END_IF;
END_REGION

REGION Network 3: Sekvens 120: Stänga av scale conveyor
   "IEC_Timer_0_DB_4".TON(IN := "Start light" AND ("Hmi_Data".Sekvensord = 120), PT := T#700MS);
   IF "IEC_Timer_0_DB_4".Q THEN
       "Conveyor Scale 0 (-)" := FALSE;
       "Hmi_Data".Sekvensord := 130;
   END_IF;
END_REGION

REGION Network 4: Sekvens 130: Väga produkten och add till totala counter om om villkoren är uppfyllda
   "IEC_Timer_0_DB_5".TON(IN := "Start light" AND ("Hmi_Data".Sekvensord = 130), PT := T#500MS);
   IF "IEC_Timer_0_DB_5".Q AND ("Skallering".IN."V är"."V ärvärde" = 12) THEN
       "Total Counter" := "Total Counter" + 1;
       "Hmi_Data"."Antal Producedrade" := "Hmi_Data"."Antal Producedrade" + 1;
       "Hmi_Data".Sekvensord := 140;
   END_IF;
   IF "IEC_Timer_0_DB_5".Q AND ("Skallering".IN."V är"."V ärvärde" <> 12) THEN
       "Hmi_Data".Sekvensord := 140;
   END_IF;
END_REGION

REGION Network 5: Sekvens 140: Stätta på och stänga av scale conveyor, removern och köra om
   #_w1 := "Start light" AND ("Hmi_Data".Sekvensord = 140);
   IF #_w1 THEN "Conveyor Scale 0 (-)" := TRUE; END_IF;
   "IEC_Timer_0_DB_6".TON(IN := #_w1 AND "Part leaving scale", PT := T#500MS);
   IF "IEC_Timer_0_DB_6".Q THEN
       "Conveyor Scale 0 (-)" := FALSE;
       "Remover 1" := FALSE;
       "Hmi_Data".Sekvensord := 0;
   END_IF;
END_REGION
END_FUNCTION

FUNCTION "ManualHmi" : Void   // FC8, LAD
{ S7_Optimized_Access := 'TRUE' }
VERSION : 0.1
   VAR_IN_OUT
      Manual : Bool;
      Output : Bool;
      Hmi : Struct
         R : Bool;
         S : Bool;
         "R light" : Bool;
         "S light" : Bool;
      END_STRUCT;
   END_VAR
BEGIN

REGION Network 1: Set och reset utgångar
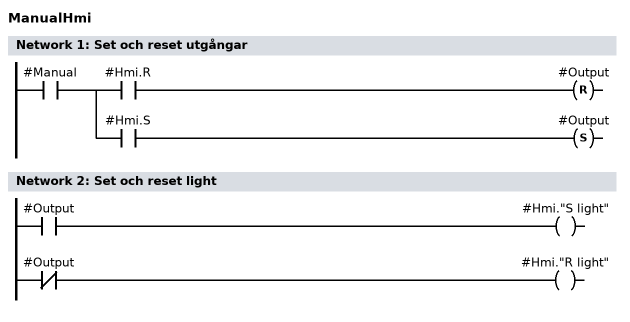
   RUNG wire#powerrail
      Contact( #Manual )
      wire#w1
      Contact( #Hmi.R )
      R_Coil( #Output )
   END_RUNG
   RUNG wire#w1
      Contact( #Hmi.S )
      S_Coil( #Output )
   END_RUNG
   // the same network as SCL:
   IF #Manual AND #Hmi.R THEN #Output := FALSE; END_IF;
   IF #Manual AND #Hmi.S THEN #Output := TRUE; END_IF;
END_REGION

REGION Network 2: Set och reset light
   RUNG wire#powerrail
      Contact( #Output )
      Coil( #Hmi."S light" )
   END_RUNG
   RUNG wire#powerrail
      I_Contact( #Output )
      Coil( #Hmi."R light" )
   END_RUNG
   // the same network as SCL:
   #Hmi."S light" := #Output;
   #Hmi."R light" := NOT #Output;
END_REGION
END_FUNCTION

FUNCTION "ManualRobot" : Void   // FC9, LAD
{ S7_Optimized_Access := 'TRUE' }
VERSION : 0.1
BEGIN

REGION Network 1: Addera/subtrahera X och Z
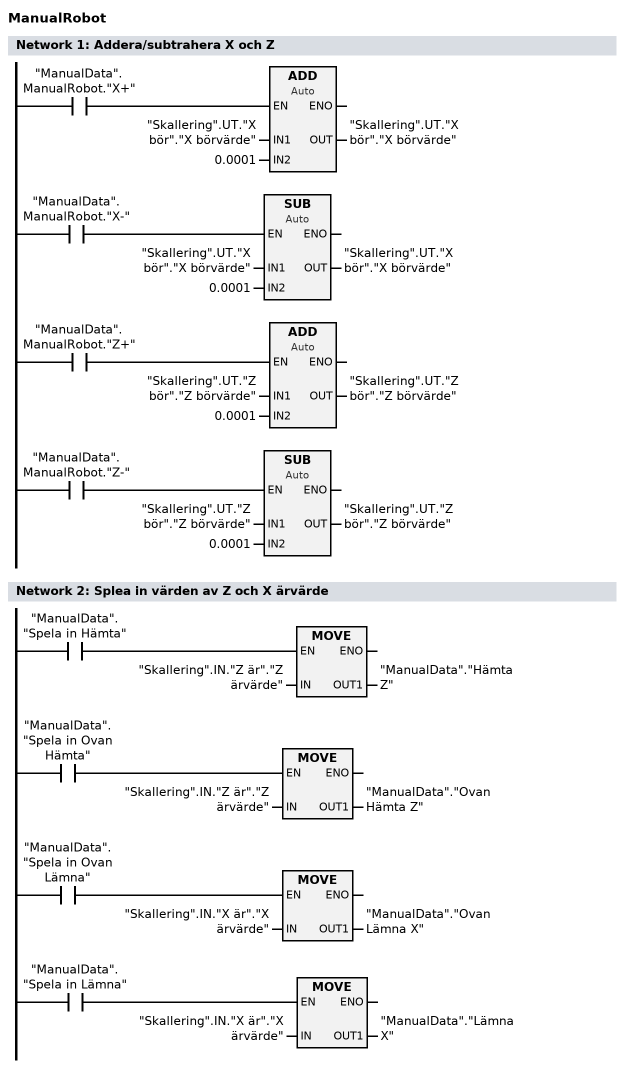
   RUNG wire#powerrail
      Contact( "ManualData".ManualRobot."X+" )
      Add(in1 := "Skallering".UT."X bör"."X börvärde", in2 := 0.0001, out => "Skallering".UT."X bör"."X börvärde")
   END_RUNG
   RUNG wire#powerrail
      Contact( "ManualData".ManualRobot."X-" )
      Sub(in1 := "Skallering".UT."X bör"."X börvärde", in2 := 0.0001, out => "Skallering".UT."X bör"."X börvärde")
   END_RUNG
   RUNG wire#powerrail
      Contact( "ManualData".ManualRobot."Z+" )
      Add(in1 := "Skallering".UT."Z bör"."Z börvärde", in2 := 0.0001, out => "Skallering".UT."Z bör"."Z börvärde")
   END_RUNG
   RUNG wire#powerrail
      Contact( "ManualData".ManualRobot."Z-" )
      Sub(in1 := "Skallering".UT."Z bör"."Z börvärde", in2 := 0.0001, out => "Skallering".UT."Z bör"."Z börvärde")
   END_RUNG
   // the same network as SCL:
   IF "ManualData".ManualRobot."X+" THEN
       "Skallering".UT."X bör"."X börvärde" := "Skallering".UT."X bör"."X börvärde" + 0.0001;
   END_IF;
   IF "ManualData".ManualRobot."X-" THEN
       "Skallering".UT."X bör"."X börvärde" := "Skallering".UT."X bör"."X börvärde" - 0.0001;
   END_IF;
   IF "ManualData".ManualRobot."Z+" THEN
       "Skallering".UT."Z bör"."Z börvärde" := "Skallering".UT."Z bör"."Z börvärde" + 0.0001;
   END_IF;
   IF "ManualData".ManualRobot."Z-" THEN
       "Skallering".UT."Z bör"."Z börvärde" := "Skallering".UT."Z bör"."Z börvärde" - 0.0001;
   END_IF;
END_REGION

REGION Network 2: Splea in värden av Z och X ärvärde
   RUNG wire#powerrail
      Contact( "ManualData"."Spela in Hämta" )
      Move(in := "Skallering".IN."Z är"."Z ärvärde", out1 => "ManualData"."Hämta Z")
   END_RUNG
   RUNG wire#powerrail
      Contact( "ManualData"."Spela in Ovan Hämta" )
      Move(in := "Skallering".IN."Z är"."Z ärvärde", out1 => "ManualData"."Ovan Hämta Z")
   END_RUNG
   RUNG wire#powerrail
      Contact( "ManualData"."Spela in Ovan Lämna" )
      Move(in := "Skallering".IN."X är"."X ärvärde", out1 => "ManualData"."Ovan Lämna X")
   END_RUNG
   RUNG wire#powerrail
      Contact( "ManualData"."Spela in Lämna" )
      Move(in := "Skallering".IN."X är"."X ärvärde", out1 => "ManualData"."Lämna X")
   END_RUNG
   // the same network as SCL:
   IF "ManualData"."Spela in Hämta" THEN
       "ManualData"."Hämta Z" := "Skallering".IN."Z är"."Z ärvärde";
   END_IF;
   IF "ManualData"."Spela in Ovan Hämta" THEN
       "ManualData"."Ovan Hämta Z" := "Skallering".IN."Z är"."Z ärvärde";
   END_IF;
   IF "ManualData"."Spela in Ovan Lämna" THEN
       "ManualData"."Ovan Lämna X" := "Skallering".IN."X är"."X ärvärde";
   END_IF;
   IF "ManualData"."Spela in Lämna" THEN
       "ManualData"."Lämna X" := "Skallering".IN."X är"."X ärvärde";
   END_IF;
END_REGION
END_FUNCTION

ORGANIZATION_BLOCK "Main"   // OB1, LAD, ProgramCycle
TITLE = "Main Program Sweep (Cycle)"
{ S7_Optimized_Access := 'TRUE' }
VERSION : 0.1
   VAR_INPUT
      Initial_Call : Bool;   // Initial call of this OB
      Remanence : Bool;   // =True, if remanent data are available
   END_VAR
   VAR_TEMP   // added for the SCL form of the ladder/FBD networks
      _w1 : Bool;
      _w2 : Bool;
      _w3 : Bool;
      _w4 : Bool;
      _w5 : Bool;
      _w6 : Bool;
      _w7 : Bool;
      _w8 : Bool;
   END_VAR
BEGIN

REGION Network 1
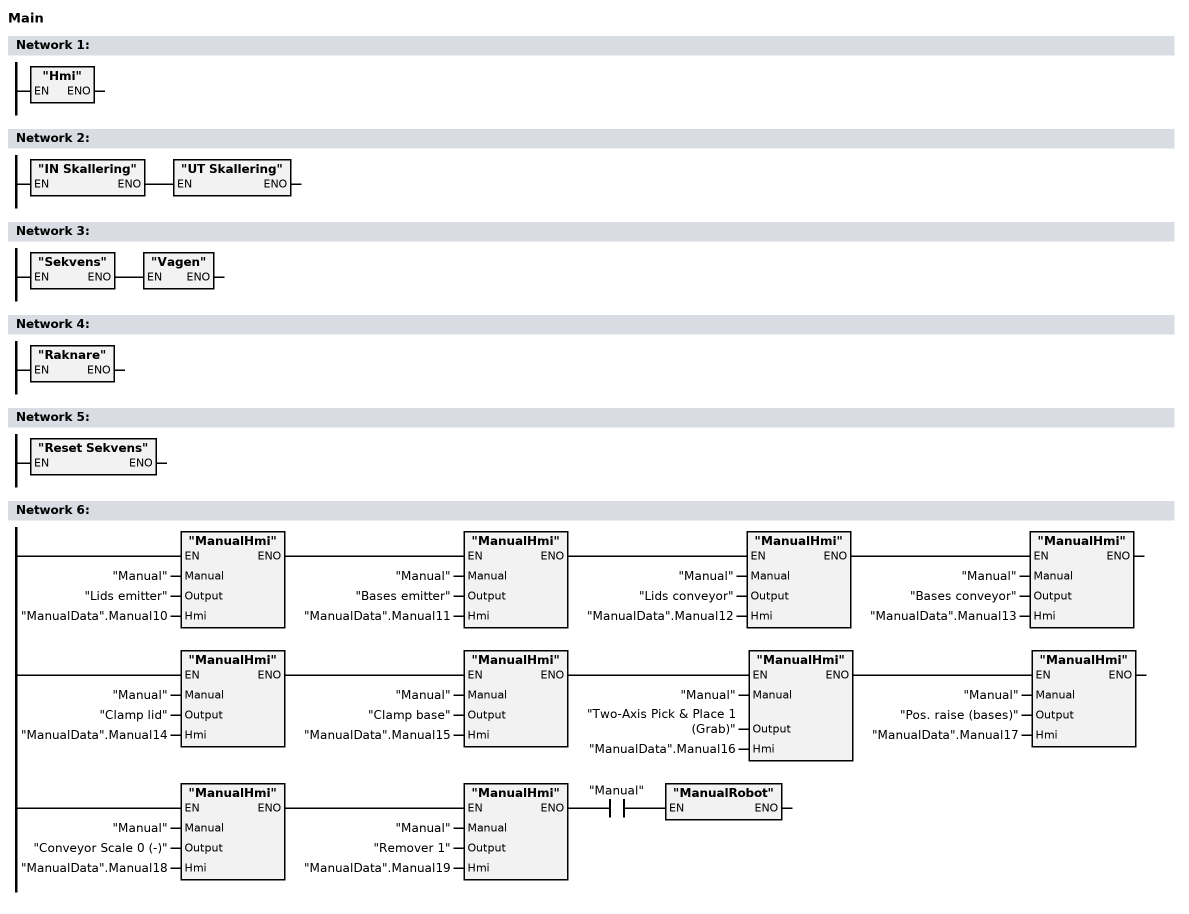
   RUNG wire#powerrail
      "Hmi"()
   END_RUNG
   // the same network as SCL:
   "Hmi"();
END_REGION

REGION Network 2
   RUNG wire#powerrail
      "IN Skallering"()
      "UT Skallering"()
   END_RUNG
   // the same network as SCL:
   "IN Skallering"(ENO => #_w1);
   IF #_w1 THEN "UT Skallering"(); END_IF;
END_REGION

REGION Network 3
   RUNG wire#powerrail
      "Sekvens"()
      "Vagen"()
   END_RUNG
   // the same network as SCL:
   "Sekvens"(ENO => #_w1);
   IF #_w1 THEN "Vagen"(); END_IF;
END_REGION

REGION Network 4
   RUNG wire#powerrail
      "Raknare"()
   END_RUNG
   // the same network as SCL:
   "Raknare"();
END_REGION

REGION Network 5
   RUNG wire#powerrail
      "Reset Sekvens"()
   END_RUNG
   // the same network as SCL:
   "Reset Sekvens"();
END_REGION

REGION Network 6
   RUNG wire#powerrail
      "ManualHmi"(Manual := "Manual", Output := "Lids emitter", Hmi := "ManualData".Manual10)
      "ManualHmi"(Manual := "Manual", Output := "Bases emitter", Hmi := "ManualData".Manual11)
      "ManualHmi"(Manual := "Manual", Output := "Lids conveyor", Hmi := "ManualData".Manual12)
      "ManualHmi"(Manual := "Manual", Output := "Bases conveyor", Hmi := "ManualData".Manual13)
   END_RUNG
   RUNG wire#powerrail
      "ManualHmi"(Manual := "Manual", Output := "Clamp lid", Hmi := "ManualData".Manual14)
      "ManualHmi"(Manual := "Manual", Output := "Clamp base", Hmi := "ManualData".Manual15)
      "ManualHmi"(Manual := "Manual", Output := "Two-Axis Pick & Place 1 (Grab)", Hmi := "ManualData".Manual16)
      "ManualHmi"(Manual := "Manual", Output := "Pos. raise (bases)", Hmi := "ManualData".Manual17)
   END_RUNG
   RUNG wire#powerrail
      "ManualHmi"(Manual := "Manual", Output := "Conveyor Scale 0 (-)", Hmi := "ManualData".Manual18)
      "ManualHmi"(Manual := "Manual", Output := "Remover 1", Hmi := "ManualData".Manual19)
      Contact( "Manual" )
      "ManualRobot"()
   END_RUNG
   // the same network as SCL:
   "ManualHmi"(Manual := "Manual", Output := "Lids emitter", Hmi := "ManualData".Manual10, ENO => #_w1);
   "ManualHmi"(EN := #_w1,
               Manual := "Manual",
               Output := "Bases emitter",
               Hmi := "ManualData".Manual11,
               ENO => #_w2);
   "ManualHmi"(EN := #_w2,
               Manual := "Manual",
               Output := "Lids conveyor",
               Hmi := "ManualData".Manual12,
               ENO => #_w3);
   IF #_w3 THEN
       "ManualHmi"(Manual := "Manual", Output := "Bases conveyor", Hmi := "ManualData".Manual13);
   END_IF;
   "ManualHmi"(Manual := "Manual", Output := "Clamp lid", Hmi := "ManualData".Manual14, ENO => #_w4);
   "ManualHmi"(EN := #_w4,
               Manual := "Manual",
               Output := "Clamp base",
               Hmi := "ManualData".Manual15,
               ENO => #_w5);
   "ManualHmi"(EN := #_w5,
               Manual := "Manual",
               Output := "Two-Axis Pick & Place 1 (Grab)",
               Hmi := "ManualData".Manual16,
               ENO => #_w6);
   IF #_w6 THEN
       "ManualHmi"(Manual := "Manual", Output := "Pos. raise (bases)", Hmi := "ManualData".Manual17);
   END_IF;
   "ManualHmi"(Manual := "Manual", Output := "Conveyor Scale 0 (-)", Hmi := "ManualData".Manual18, ENO => #_w7);
   "ManualHmi"(EN := #_w7, Manual := "Manual", Output := "Remover 1", Hmi := "ManualData".Manual19, ENO => #_w8);
   IF #_w8 AND "Manual" THEN "ManualRobot"(); END_IF;
END_REGION
END_ORGANIZATION_BLOCK

(* ===== HMI "HMI_RT_1" =====
system functions are stored by id; their names below are inferred from use
connection "HMI_Connection_1": ETHERNET, SMART_S7_1500_OMS

HMI tags "Default tag table"
   "Tag_ScreenNumber" : UInt, internal
   "Hmi_Data_Start" : Bool = PLC Hmi_Data.Start, 1 s
   "Hmi_Data_Stop" : Bool = PLC Hmi_Data.Stop, 1 s
   "Hmi_Data_Reset" : Bool = PLC Hmi_Data.Reset, 1 s
   "Hmi_Data_Sekvensord" : Int = PLC Hmi_Data.Sekvensord, 100 ms
   "Hmi_Data_Reset Sekvens" : Int = PLC Hmi_Data."Reset Sekvens", 100 ms
   "Hmi_Data_Beställning" : Int = PLC Hmi_Data.Beställning, 1 s
   "Hmi_Data_Antal Producedrade" : Int = PLC Hmi_Data."Antal Producedrade", 100 ms
   "Hmi_Data_Order" : Bool = PLC Hmi_Data.Order, 1 s
   "Weight" : Int = PLC Weight AT %QW36, 100 ms
   "GB&GL" : Int = PLC "GB&GL" AT %QW38, 1 s
   "GB&BL" : Int = PLC "GB&BL" AT %QW42, 1 s
   "BB&GL" : Int = PLC "BB&GL" AT %QW44, 1 s
   "BB&BL" : Int = PLC "BB&BL" AT %QW40, 1 s
   "Total Counter" : Int = PLC "Total Counter" AT %QW30, 100 ms
   "ManualData_Manual10_R" : Bool = PLC ManualData.Manual10.R, 1 s
   "ManualData_Manual10_R light" : Bool = PLC ManualData.Manual10."R light", 1 s
   "ManualData_Manual10_S light" : Bool = PLC ManualData.Manual10."S light", 1 s
   "ManualData_Manual10_S" : Bool = PLC ManualData.Manual10.S, 1 s
   "ManualData_Manual11_R light" : Bool = PLC ManualData.Manual11."R light", 1 s
   "ManualData_Manual11_R" : Bool = PLC ManualData.Manual11.R, 1 s
   "ManualData_Manual12_R" : Bool = PLC ManualData.Manual12.R, 1 s
   "ManualData_Manual13_R" : Bool = PLC ManualData.Manual13.R, 1 s
   "ManualData_Manual14_R" : Bool = PLC ManualData.Manual14.R, 1 s
   "ManualData_Manual11_S" : Bool = PLC ManualData.Manual11.S, 1 s
   "ManualData_Manual12_S" : Bool = PLC ManualData.Manual12.S, 1 s
   "ManualData_Manual13_S" : Bool = PLC ManualData.Manual13.S, 1 s
   "ManualData_Manual14_S" : Bool = PLC ManualData.Manual14.S, 1 s
   "ManualData_Manual11_S light" : Bool = PLC ManualData.Manual11."S light", 1 s
   "ManualData_Manual12_S light" : Bool = PLC ManualData.Manual12."S light", 1 s
   "ManualData_Manual13_S light" : Bool = PLC ManualData.Manual13."S light", 1 s
   "ManualData_Manual14_S light" : Bool = PLC ManualData.Manual14."S light", 1 s
   "ManualData_Manual14_R light" : Bool = PLC ManualData.Manual14."R light", 1 s
   "ManualData_Manual13_R light" : Bool = PLC ManualData.Manual13."R light", 1 s
   "ManualData_Manual12_R light" : Bool = PLC ManualData.Manual12."R light", 1 s
   "ManualData_Manual15_R" : Bool = PLC ManualData.Manual15.R, 1 s
   "ManualData_Manual15_S" : Bool = PLC ManualData.Manual15.S, 1 s
   "ManualData_Manual15_R light" : Bool = PLC ManualData.Manual15."R light", 1 s
   "ManualData_Manual15_S light" : Bool = PLC ManualData.Manual15."S light", 1 s
   "Lid at place" : Bool = PLC "Lid at place" AT %I0.3, 100 ms
   "Base at place" : Bool = PLC "Base at place" AT %I0.6, 100 ms
   "Two-Axis Pick & Place 1 (Item Detected)" : Bool = PLC "Two-Axis Pick & Place 1 (Item Detected)" AT %I2.2, 100 ms
   "Part leaving" : Bool = PLC "Part leaving" AT %I1.1, 100 ms
   "Part at scale" : Bool = PLC "Part at scale" AT %I2.4, 100 ms
   "Part leaving scale" : Bool = PLC "Part leaving scale" AT %I2.5, 100 ms
   "ManualData_Manual16_R light" : Bool = PLC ManualData.Manual16."R light", 1 s
   "ManualData_Manual16_S light" : Bool = PLC ManualData.Manual16."S light", 1 s
   "ManualData_Manual16_R" : Bool = PLC ManualData.Manual16.R, 1 s
   "ManualData_Manual16_S" : Bool = PLC ManualData.Manual16.S, 1 s
   "ManualData_Manual17_R" : Bool = PLC ManualData.Manual17.R, 1 s
   "ManualData_Manual17_S" : Bool = PLC ManualData.Manual17.S, 1 s
   "ManualData_Manual17_S light" : Bool = PLC ManualData.Manual17."S light", 1 s
   "ManualData_Manual17_R light" : Bool = PLC ManualData.Manual17."R light", 1 s
   "ManualData_Manual18_R" : Bool = PLC ManualData.Manual18.R, 1 s
   "ManualData_Manual18_S" : Bool = PLC ManualData.Manual18.S, 1 s
   "ManualData_Manual18_S light" : Bool = PLC ManualData.Manual18."S light", 1 s
   "ManualData_Manual18_R light" : Bool = PLC ManualData.Manual18."R light", 1 s
   "Auto" : Bool = PLC Auto AT %I1.7, 1 s
   "Manual" : Bool = PLC Manual AT %I1.6, 1 s
   "Skallering_IN_X är_X ärvärde" : Real = PLC Skallering.IN."X är"."X ärvärde", 100 ms
   "Skallering_IN_Z är_Z ärvärde" : Real = PLC Skallering.IN."Z är"."Z ärvärde", 100 ms
   "Skallering_UT_X bör_X börvärde" : Real = PLC Skallering.UT."X bör"."X börvärde", 100 ms
   "Skallering_UT_Z bör_Z börvärde" : Real = PLC Skallering.UT."Z bör"."Z börvärde", 100 ms
   "ManualData_Manual19_R" : Bool = PLC ManualData.Manual19.R, 1 s
   "ManualData_Manual19_S" : Bool = PLC ManualData.Manual19.S, 1 s
   "ManualData_Manual19_R light" : Bool = PLC ManualData.Manual19."R light", 1 s
   "ManualData_Manual19_S light" : Bool = PLC ManualData.Manual19."S light", 1 s
   "ManualData_ManualRobot_Z+" : Bool = PLC ManualData.ManualRobot.Z+, 1 s
   "ManualData_ManualRobot_X-" : Bool = PLC ManualData.ManualRobot.X-, 1 s
   "ManualData_ManualRobot_Z-" : Bool = PLC ManualData.ManualRobot.Z-, 1 s
   "ManualData_ManualRobot_X+" : Bool = PLC ManualData.ManualRobot.X+, 1 s
   "ManualData_Spela in Hämta" : Bool = PLC ManualData."Spela in Hämta", 1 s
   "ManualData_Spela in Ovan Hämta" : Bool = PLC ManualData."Spela in Ovan Hämta", 1 s
   "ManualData_Spela in Ovan Lämna" : Bool = PLC ManualData."Spela in Ovan Lämna", 1 s
   "ManualData_Spela in Lämna" : Bool = PLC ManualData."Spela in Lämna", 1 s

text list "Sekvensord": 0 'Sekvens 0: Sätta igång emitters och conveyors'; 10 'Sekvens 10: Sätta igång clamperna och stänga av conveyors'; 20 'Sekvens 20: Dra ner armen och stänga av clamperna'; 30 'Sekvens 30: Sätta igång Grab'; 40 'Sekvens 40: Dra up armen'; 50 'Sekvens 50: Dra ut armen'; 60 'Sekvens 60: Dra ner armen'; 70 'Sekvens 70: Stänga av Grab och dra up armen'; 80 'Sekvens 80: Dra in armen och stätta igång Pos. raise, conveyors och stänga av emittrarna'; 90 'Sekvens 90: Stänga av Pos. raise'; 100 'Sekvens 100: Stätta på scale conveyor och removern'; 110 'Sekvens 110: Stänga av conveyors'; 120 'Sekvens 120: Stänga av scale conveyor'; 130 'Sekvens 130: Väga produkten och add till totala counter om om villkoren är uppfyllda'; 140 'Sekvens 140: Stätta på och stänga av scale conveyor, removern och köra om'

text list "Reset Sekvens": 0 'Sekvens 0: Skicka 100 till Reset Sekvensen om Grab är på annars skicka 10'; 10 'Sekvens 10: Dra up armen'; 20 'Sekvens 20: Dra tillbaka armen'; 30 'Sekvens 30: Sätta på Conveyors, Pos. raisers och Removers'; 40 'Sekvens 40: Stänga av Conveyors, Pos. raisers och Removers'; 100 'Sekvens 100: Dra up armen (om Grab är på)'; 110 'Sekvens 110: Dra tillbaka armen (om Grab är på)'; 120 'Sekvens 120: Dra ner armen (om Grab är på)'; 130 'Sekvens 130: Stänga av Grab, dra up armen och kör Sekvens 30 igen'

screen "Root screen" 800x480, template "Template_1"
   on GenerateScreen: SetTag("Tag_ScreenNumber", 1)
   TextField "HmiScreenItemData_3" at 105,199 size 640x25; Text 'Welcome to HMI_1 (KTP700 Basic+ PN)!'
   Button "HmiScreenItemData" at 31,83 size 159x47; TextOff 'StartStop'; PictureOff "Navigates to StartStop for KTP700 Basic+ PN 17.0.0.0"; PictureOn "Navigates to StartStop for KTP700 Basic+ PN 17.0.0.0"
      on Release: ActivateScreen("StartStop", 0)
   Button "HmiScreenItemData_1" at 32,195 size 159x47; TextOff 'Statistik'; PictureOff "Navigates to Statistik for KTP700 Basic+ PN 17.0.0.0"; PictureOn "Navigates to Statistik for KTP700 Basic+ PN 17.0.0.0"
      on Release: ActivateScreen("Statistik", 0)
   Button "HmiScreenItemData_2" at 32,140 size 159x47; TextOff 'Info&Beställning'; PictureOff "Navigates to Info&Beställning for KTP700 Basic+ PN 17.0.0.0"; PictureOn "Navigates to Info&Beställning for KTP700 Basic+ PN 17.0.0.0"
      on Release: ActivateScreen("Info&Beställning", 0)
   Button "HmiScreenItemData_4" at 33,365 size 159x47; TextOff 'System screens'; PictureOff "Navigates to System screens for KTP700 Basic+ PN 17.0.0.0"; PictureOn "Navigates to System screens for KTP700 Basic+ PN 17.0.0.0"
      on Release: ActivateScreen("System screens", 0)
   Button "Button_1" at 32,251 size 159x47; TextOff 'Manual'; PictureOff "Navigates to Info&Beställning for KTP700 Basic+ PN 17.0.0.0"; PictureOn "Navigates to Info&Beställning for KTP700 Basic+ PN 17.0.0.0"
      on Click: ActivateScreen("Manual", 0)
   Button "Button_2" at 32,309 size 159x47; TextOff 'Manual Robot'; PictureOff "Navigates to Info&Beställning for KTP700 Basic+ PN 17.0.0.0"; PictureOn "Navigates to Info&Beställning for KTP700 Basic+ PN 17.0.0.0"
      on Click: ActivateScreen("Manual Robot", 0)

screen "StartStop" 800x480, template "Template_1"
   on GenerateScreen: SetTag("Tag_ScreenNumber", 2)
   TextField "HmiScreenItemData" at 0,6 size 160x46; Text 'Start Stop'
   Button "Back" at 1,52 size 159x46; TextOff 'Tillbaka'; TextOn 'Back'
      on Release: ActivateScreen("Root screen", 0)
   Button "Button_1" at 122,182 size 130x60; TextOff 'Start knapp'
      on Press: function_b14e0dd5("Hmi_Data_Start", 0)
   Button "Button_2" at 539,182 size 130x60; TextOff 'Stop knapp'
      on Press: function_b14e0dd5("Hmi_Data_Stop", 0)
   Button "Button_3" at 331,182 size 130x60; TextOff 'Reset knapp'
      on Press: function_b14e0dd5("Hmi_Data_Reset", 0)

screen "Statistik" 800x480, template "Template_1"
   on GenerateScreen: SetTag("Tag_ScreenNumber", 3)
   TextField "HmiScreenItemData" at 0,4 size 148x46; Text 'Statistik'
   IOField "I/O field_1" at 603,233 size 82x32; FormatPattern 999; Unit  KG
      ProcessValue <- "Weight"
   IOField "I/O field_2" at 90,201 size 96x32; FormatPattern 9999
      ProcessValue <- "GB&GL"
   IOField "I/O field_3" at 353,201 size 96x32; FormatPattern 9999
      ProcessValue <- "GB&BL"
   IOField "I/O field_4" at 353,314 size 96x32; FormatPattern 9999
      ProcessValue <- "BB&GL"
   IOField "I/O field_5" at 90,314 size 96x32; FormatPattern 9999
      ProcessValue <- "BB&BL"
   IOField "I/O field_6" at 543,282 size 221x32; FormatPattern 9999; Unit  Totalt Producerade
      ProcessValue <- "Total Counter"
   TextField "Text field_2" at 18,167 size 96x28; Text 'Grån Bas'
   TextField "Text field_3" at 27,276 size 79x28; Text 'Blå Bas'
   TextField "Text field_7" at 116,167 size 21x28; Text '&'
   TextField "Text field_8" at 113,276 size 21x28; Text '&'
   TextField "Text field_4" at 137,276 size 73x28; Text 'Blå Lid'
   TextField "Text field_5" at 144,167 size 90x28; Text 'Grån Lid'
   TextField "Text field_6" at 292,167 size 96x28; Text 'Grån Bas'
   TextField "Text field_9" at 391,167 size 21x28; Text '&'
   TextField "Text field_10" at 419,167 size 73x28; Text 'Blå Lid'
   TextField "Text field_11" at 419,276 size 90x28; Text 'Grån Lid'
   TextField "Text field_12" at 396,278 size 21x28; Text '&'
   TextField "Text field_13" at 312,276 size 79x28; Text 'Blå Bas'
   Button "Back" at 1,52 size 159x46; TextOn 'Back'; TextOff 'Tillbaka'
      on Release: ActivateScreen("Root screen", 0)

screen "Info&Beställning" 800x480, template "Template_1"
   on GenerateScreen: SetTag("Tag_ScreenNumber", 4)
   TextField "HmiScreenItemData" at 12,6 size 229x46; Text 'Info & Beställning'
   IOField "I/O field_1" at 21,262 size 96x32; FormatPattern 9999
      ProcessValue <- "Hmi_Data_Sekvensord"
   IOField "I/O field_2" at 190,263 size 96x32; FormatPattern 9999
      ProcessValue <- "Hmi_Data_Reset Sekvens"
   SymbolicIOField "Symbolic I/O field_1" at 20,321 size 753x32; TextOff '0'; TextOn '1'; TextList "Sekvensord"
      ProcessValue <- "Hmi_Data_Sekvensord"
   SymbolicIOField "Symbolic I/O field_2" at 21,368 size 753x32; TextOn '1'; TextOff '0'; TextList "Reset Sekvens"
      ProcessValue <- "Hmi_Data_Reset Sekvens"
   IOField "I/O field_3" at 555,213 size 217x32; FormatPattern 9999; Unit  Antal Beställda
      ProcessValue <- "Hmi_Data_Beställning"
   IOField "I/O field_4" at 556,263 size 217x32; FormatPattern 9999; Unit  Antal Producerade
      ProcessValue <- "Hmi_Data_Antal Producedrade"
   Button "Button_1" at 618,155 size 96x32; TextOff 'Order'
      on Press: InvertBit("Hmi_Data_Order")
   Circle "Circle_1" at 643,96 size 39x39
      Appearance <- "Hmi_Data_Order"
   Button "Back" at 1,52 size 159x46; TextOn 'Back'; TextOff 'Tillbaka'
      on Release: ActivateScreen("Root screen", 0)

screen "System screens" 800x480, template "Template_1"
   on GenerateScreen: SetTag("Tag_ScreenNumber", 5)
   Button "Back" at 1,52 size 159x47; TextOff 'Back'
      on Release: ActivateScreen("Root screen", 0)
   Button "HmiScreenItemData" at 36,146 size 159x47; TextOff 'User administration'; PictureOff "Navigates to User administration for KTP700 Basic+ PN 17.0.0.0"; PictureOn "Navigates to User administration for KTP700 Basic+ PN 17.0.0.0"
      on Release: ActivateScreen("User administration", 0)
   Button "HmiScreenItemData_1" at 36,205 size 159x47; TextOff 'Different jobs'; PictureOff "Navigates to Different jobs for KTP700 Basic+ PN 17.0.0.0"; PictureOn "Navigates to Different jobs for KTP700 Basic+ PN 17.0.0.0"
      on Release: ActivateScreen("Different jobs", 0)

screen "User administration" 800x480, template "Template_1"
   on GenerateScreen: SetTag("Tag_ScreenNumber", 6)
   UserView "HmiScreenItemData" at 1,100 size 796x321
   Button "Back" at 1,52 size 159x47; TextOff 'Back'
      on Release: ActivateScreen("System screens", 0)

screen "Different jobs" 800x480, template "Template_1"
   on GenerateScreen: SetTag("Tag_ScreenNumber", 7)
   Button "Toggle language" at 36,146 size 159x47; TextOff 'Toggle language'
      on Release: function_fb9197e8(-1)
   Button "Back" at 1,52 size 159x47; TextOff 'Back'
      on Release: ActivateScreen("System screens", 0)

screen "Manual" 800x480
   TextField "Text field_1" at 18,6 size 103x37; Text 'Manuel'
   Button "Button_1" at 31,152 size 80x40; TextOff 'R'
      on Press: function_b14e0dd5("ManualData_Manual10_R", 0)
      Appearance <- "ManualData_Manual10_R light"
   Button "Button_2" at 143,152 size 80x40; TextOff 'S'
      on Press: function_b14e0dd5("ManualData_Manual10_S", 0)
      Appearance <- "ManualData_Manual10_S light"
   Button "Button_3" at 31,245 size 80x40; TextOff 'R'
      on Press: function_b14e0dd5("ManualData_Manual11_R", 0)
      Appearance <- "ManualData_Manual11_R light"
   Button "Button_4" at 31,330 size 80x40; TextOff 'R'
      on Press: function_b14e0dd5("ManualData_Manual12_R", 0)
      Appearance <- "ManualData_Manual12_R light"
   Button "Button_5" at 32,409 size 80x40; TextOff 'R'
      on Press: function_b14e0dd5("ManualData_Manual13_R", 0)
      Appearance <- "ManualData_Manual13_R light"
   Button "Button_6" at 262,152 size 80x40; TextOff 'R'
      on Press: function_b14e0dd5("ManualData_Manual14_R", 0)
      Appearance <- "ManualData_Manual14_R light"
   Button "Button_7" at 143,244 size 80x40; TextOff 'S'
      on Press: function_b14e0dd5("ManualData_Manual11_S", 0)
      Appearance <- "ManualData_Manual11_S light"
   Button "Button_8" at 143,329 size 80x40; TextOff 'S'
      on Press: function_b14e0dd5("ManualData_Manual12_S", 0)
      Appearance <- "ManualData_Manual12_S light"
   Button "Button_9" at 142,410 size 80x40; TextOff 'S'
      on Press: function_b14e0dd5("ManualData_Manual13_S", 0)
      Appearance <- "ManualData_Manual13_S light"
   Button "Button_10" at 378,152 size 80x40; TextOff 'S'
      on Press: function_b14e0dd5("ManualData_Manual14_S", 0)
      Appearance <- "ManualData_Manual14_S light"
   TextField "Text field_2" at 57,120 size 121x27; Text 'Lids Emitter'
   TextField "Text field_3" at 49,215 size 137x27; Text 'Bases Emitter'
   TextField "Text field_4" at 49,300 size 140x27; Text 'Lids Conveyor'
   TextField "Text field_5" at 45,381 size 156x27; Text 'Bases Conveyor'
   Button "Button_11" at 262,244 size 80x40; TextOff 'R'
      on Press: function_b14e0dd5("ManualData_Manual15_R", 0)
      Appearance <- "ManualData_Manual15_R light"
   Button "Button_12" at 378,244 size 80x40; TextOff 'S'
      on Press: function_b14e0dd5("ManualData_Manual15_S", 0)
      Appearance <- "ManualData_Manual15_S light"
   TextField "Text field_6" at 302,120 size 100x27; Text 'Clamp Lid'
   TextField "Text field_7" at 302,217 size 116x27; Text 'Clamp Base'
   Circle "Circle_1" at 689,248 size 39x39
      Appearance <- "Part leaving scale"
   Circle "Circle_2" at 533,163 size 39x39
      Appearance <- "Two-Axis Pick & Place 1 (Item Detected)"
   Circle "Circle_3" at 532,70 size 39x39
      Appearance <- "Lid at place"
   Circle "Circle_4" at 533,248 size 39x39
      Appearance <- "Part at scale"
   Circle "Circle_5" at 689,163 size 39x39
      Appearance <- "Part leaving"
   Circle "Circle_6" at 689,70 size 39x39
      Appearance <- "Base at place"
   TextField "Text field_8" at 498,43 size 103x25; Text 'Lid at place'
   TextField "Text field_9" at 651,43 size 118x25; Text 'Base at place'
   TextField "Text field_10" at 487,137 size 128x25; Text 'Item Detected'
   TextField "Text field_11" at 655,137 size 107x25; Text 'Part leaving'
   TextField "Text field_12" at 494,223 size 110x25; Text 'Part at scale'
   TextField "Text field_14" at 635,223 size 155x25; Text 'Part leaving scale'
   Button "Button_13" at 262,409 size 80x40; TextOff 'R'
      on Press: function_b14e0dd5("ManualData_Manual17_R", 0)
      Appearance <- "ManualData_Manual17_R light"
   Button "Button_14" at 378,409 size 80x40; TextOff 'S'
      on Press: function_b14e0dd5("ManualData_Manual17_S", 0)
      Appearance <- "ManualData_Manual17_S light"
   TextField "Text field_13" at 272,380 size 175x27; Text 'Pos. raise (bases)'
   Button "Button_15" at 529,328 size 80x40; TextOff 'R'
      on Press: function_b14e0dd5("ManualData_Manual18_R", 0)
      Appearance <- "ManualData_Manual18_R light"
   Button "Button_16" at 645,328 size 80x40; TextOff 'S'
      on Press: function_b14e0dd5("ManualData_Manual18_S", 0)
      Appearance <- "ManualData_Manual18_S light"
   TextField "Text field_15" at 524,300 size 201x27; Text 'Conveyor Scale 0 (-)'
   Button "Button_17" at 528,407 size 80x40; TextOff 'R'
      on Press: function_b14e0dd5("ManualData_Manual19_R", 0)
      Appearance <- "ManualData_Manual19_R light"
   Button "Button_18" at 644,408 size 80x40; TextOff 'S'
      on Press: function_b14e0dd5("ManualData_Manual19_S", 0)
      Appearance <- "ManualData_Manual19_S light"
   TextField "Text field_16" at 573,378 size 108x27; Text 'Remover 1'
   Button "Button_19" at 262,327 size 80x40; TextOff 'R'
      on Press: function_b14e0dd5("ManualData_Manual16_R", 0)
      Appearance <- "ManualData_Manual16_R light"
   Button "Button_20" at 378,327 size 80x40; TextOff 'S'
      on Press: function_b14e0dd5("ManualData_Manual16_S", 0)
      Appearance <- "ManualData_Manual16_S light"
   TextField "Text field_17" at 329,299 size 50x27; Text 'Grab'
   Button "Back" at 1,52 size 159x46; TextOn 'Back'; TextOff 'Tillbaka'
      on Release: ActivateScreen("Root screen", 0)

screen "Manual Robot" 800x480
   TextField "Text field_1" at 12,8 size 193x37; Text 'Manual Robot'
   IOField "I/O field_1" at 156,117 size 115x32; FormatPattern s99999.999
      ProcessValue <- "Skallering_IN_X är_X ärvärde"
   IOField "I/O field_2" at 334,117 size 115x32; FormatPattern s99999.999
      ProcessValue <- "Skallering_IN_Z är_Z ärvärde"
   TextField "Text field_2" at 186,87 size 38x23; Text 'X är'
   TextField "Text field_3" at 371,87 size 37x23; Text 'Z är'
   IOField "I/O field_3" at 156,200 size 115x32; FormatPattern s99999.999
      ProcessValue <- "Skallering_UT_X bör_X börvärde"
   TextField "Text field_4" at 186,173 size 48x23; Text 'X bör'
   IOField "I/O field_4" at 334,200 size 115x32; FormatPattern s99999.999
      ProcessValue <- "Skallering_UT_Z bör_Z börvärde"
   TextField "Text field_5" at 371,170 size 47x23; Text 'Z bör'
   Circle "Circle_1" at 684,117 size 39x39
      Appearance <- "Manual"
   TextField "Text field_6" at 670,85 size 64x23; Text 'Manual'
   Button "Button_1" at 255,379 size 96x32; TextOff 'Z+'
      on Press: function_b14e0dd5("ManualData_ManualRobot_Z+", 0)
   Button "Button_2" at 131,318 size 96x32; TextOff 'X+'
      on Press: function_b14e0dd5("ManualData_ManualRobot_X+", 0)
   Button "Button_3" at 376,318 size 96x32; TextOff 'X-'
      on Press: function_b14e0dd5("ManualData_ManualRobot_X-", 0)
   Button "Button_4" at 254,259 size 96x32; TextOff 'Z-'
      on Press: function_b14e0dd5("ManualData_ManualRobot_Z-", 0)
   Button "Button_5" at 599,228 size 185x32; TextOff 'Spela in Hämta'
      on Press: function_b14e0dd5("ManualData_Spela in Hämta", 0)
   Button "Button_6" at 600,286 size 185x32; TextOff 'Splea in Ovan Hämta'
      on Press: function_b14e0dd5("ManualData_Spela in Ovan Hämta", 0)
   Button "Button_7" at 600,341 size 185x32; TextOff 'Spela in Ovan Lämna'
      on Press: function_b14e0dd5("ManualData_Spela in Ovan Lämna", 0)
   Button "Button_8" at 601,395 size 185x32; TextOff 'Spela in Lämna'
      on Press: function_b14e0dd5("ManualData_Spela in Lämna", 0)
   Button "Back" at 1,52 size 159x46; TextOn 'Back'; TextOff 'Tillbaka'
      on Release: ActivateScreen("Root screen", 0)
*)